LIN {X 0,Y 566.216,Z 387.456,A -85,B 0,C 180,E1 -2672.661,E2 -2672.661} C_VEL
LIN {X 0,Y 566.231,Z 387.453,A -85,B 0,C 180,E1 -2675.038,E2 -2675.038} C_VEL
LIN {X 0,Y 566.19,Z 387.454,A -85,B 0,C 180,E1 -2678.137,E2 -2678.137} C_VEL
LIN {X 0,Y 566.23,Z 387.456,A -85,B 0,C 180,E1 -2680.611,E2 -2680.611} C_VEL
LIN {X 0,Y 566.216,Z 387.449,A -85,B 0,C 180,E1 -2683.412,E2 -2683.412} C_VEL
LIN {X 0,Y 566.196,Z 387.457,A -85,B 0,C 180,E1 -2686.358,E2 -2686.358} C_VEL
LIN {X 0,Y 566.228,Z 387.456,A -85,B 0,C 180,E1 -2688.675,E2 -2688.675} C_VEL
LIN {X 0,Y 566.229,Z 387.447,A -85,B 0,C 180,E1 -2691.434,E2 -2691.434} C_VEL
LIN {X 0,Y 566.256,Z 387.451,A -85,B 0,C 180,E1 -2694.301,E2 -2694.301} C_VEL
LIN {X 0,Y 566.275,Z 387.444,A -85,B 0,C 180,E1 -2697.866,E2 -2697.866} C_VEL
LIN {X 0,Y 566.299,Z 387.443,A -85,B 0,C 180,E1 -2700.711,E2 -2700.711} C_VEL
LIN {X 0,Y 566.27,Z 387.445,A -85,B 0,C 180,E1 -2702.845,E2 -2702.845} C_VEL
LIN {X 0,Y 566.256,Z 387.446,A -85,B 0,C 180,E1 -2705.698,E2 -2705.698} C_VEL
LIN {X 0,Y 566.228,Z 387.452,A -85,B 0,C 180,E1 -2708.565,E2 -2708.565} C_VEL
LIN {X 0,Y 566.234,Z 387.447,A -85,B 0,C 180,E1 -2711.454,E2 -2711.454} C_VEL
LIN {X 0,Y 566.227,Z 387.452,A -85,B 0,C 180,E1 -2714.507,E2 -2714.507} C_VEL
LIN {X 0,Y 566.197,Z 387.452,A -85,B 0,C 180,E1 -2717.331,E2 -2717.331} C_VEL
LIN {X 0,Y 566.207,Z 387.456,A -85,B 0,C 180,E1 -2720.337,E2 -2720.337} C_VEL
LIN {X 0,Y 566.182,Z 387.455,A -85,B 0,C 180,E1 -2723.404,E2 -2723.404} C_VEL
LIN {X 0,Y 566.217,Z 387.455,A -85,B 0,C 180,E1 -2725.748,E2 -2725.748} C_VEL
LIN {X 0,Y 566.211,Z 387.451,A -85,B 0,C 180,E1 -2727.49,E2 -2727.49} C_VEL
LIN {X 0,Y 565.532,Z 387.542,A -85,B 0,C 180,E1 -2728.084,E2 -2728.084} C_VEL
LIN {X 0,Y 562.666,Z 387.896,A -85,B 0,C 180,E1 -2729.047,E2 -2729.047} C_VEL
LIN {X 0,Y 560.255,Z 388.2,A -85,B 0,C 180,E1 -2729.823,E2 -2729.823} C_VEL
LIN {X 0,Y 559.226,Z 388.322,A -85,B 0,C 180,E1 -2730.422,E2 -2730.422} C_VEL
LIN {X 0,Y 559.145,Z 388.331,A -85,B 0,C 180,E1 -2730.624,E2 -2730.624} C_VEL
LIN {X 0,Y 559.171,Z 388.332,A -85,B 0,C 180,E1 -2733.574,E2 -2733.574} C_VEL
LIN {X 0,Y 559.162,Z 388.329,A -85,B 0,C 180,E1 -2736.449,E2 -2736.449} C_VEL
LIN {X 0,Y 559.172,Z 388.327,A -85,B 0,C 180,E1 -2738.934,E2 -2738.934} C_VEL
LIN {X 0,Y 559.185,Z 388.335,A -85,B 0,C 180,E1 -2741.768,E2 -2741.768} C_VEL
LIN {X 0,Y 559.133,Z 388.331,A -85,B 0,C 180,E1 -2744.739,E2 -2744.739} C_VEL
LIN {X 0,Y 559.161,Z 388.331,A -85,B 0,C 180,E1 -2747.258,E2 -2747.258} C_VEL
LIN {X 0,Y 559.179,Z 388.328,A -85,B 0,C 180,E1 -2750.135,E2 -2750.135} C_VEL
LIN {X 0,Y 559.14,Z 388.331,A -85,B 0,C 180,E1 -2752.892,E2 -2752.892} C_VEL
LIN {X 0,Y 559.155,Z 388.338,A -85,B 0,C 180,E1 -2755.557,E2 -2755.557} C_VEL
LIN {X 0,Y 559.166,Z 388.328,A -85,B 0,C 180,E1 -2758.138,E2 -2758.138} C_VEL
LIN {X 0,Y 559.139,Z 388.331,A -85,B 0,C 180,E1 -2760.647,E2 -2760.647} C_VEL
LIN {X 0,Y 559.177,Z 388.332,A -85,B 0,C 180,E1 -2763.17,E2 -2763.17} C_VEL
LIN {X 0,Y 559.153,Z 388.337,A -85,B 0,C 180,E1 -2765.495,E2 -2765.495} C_VEL
LIN {X 0,Y 559.167,Z 388.328,A -85,B 0,C 180,E1 -2768.624,E2 -2768.624} C_VEL
LIN {X 0,Y 559.165,Z 388.331,A -85,B 0,C 180,E1 -2770.927,E2 -2770.927} C_VEL
LIN {X 0,Y 559.163,Z 388.33,A -85,B 0,C 180,E1 -2773.948,E2 -2773.948} C_VEL
LIN {X 0,Y 559.169,Z 388.328,A -85,B 0,C 180,E1 -2776.184,E2 -2776.184} C_VEL
LIN {X 0,Y 559.193,Z 388.334,A -85,B 0,C 180,E1 -2779.134,E2 -2779.134} C_VEL
LIN {X 0,Y 559.203,Z 388.324,A -85,B 0,C 180,E1 -2782.054,E2 -2782.054} C_VEL
LIN {X 0,Y 559.253,Z 388.325,A -85,B 0,C 180,E1 -2784.954,E2 -2784.954} C_VEL
LIN {X 0,Y 559.254,Z 388.318,A -85,B 0,C 180,E1 -2787.84,E2 -2787.84} C_VEL
LIN {X 0,Y 559.27,Z 388.321,A -85,B 0,C 180,E1 -2790.72,E2 -2790.72} C_VEL
LIN {X 0,Y 559.236,Z 388.328,A -85,B 0,C 180,E1 -2792.882,E2 -2792.882} C_VEL
LIN {X 0,Y 559.236,Z 388.32,A -85,B 0,C 180,E1 -2795.77,E2 -2795.77} C_VEL
LIN {X 0,Y 559.189,Z 388.332,A -85,B 0,C 180,E1 -2798.674,E2 -2798.674} C_VEL
LIN {X 0,Y 559.202,Z 388.324,A -85,B 0,C 180,E1 -2801.6,E2 -2801.6} C_VEL
LIN {X 0,Y 559.197,Z 388.331,A -85,B 0,C 180,E1 -2804.596,E2 -2804.596} C_VEL
LIN {X 0,Y 559.156,Z 388.33,A -85,B 0,C 180,E1 -2807.557,E2 -2807.557} C_VEL
LIN {X 0,Y 559.169,Z 388.327,A -85,B 0,C 180,E1 -2809.837,E2 -2809.837} C_VEL
LIN {X 0,Y 559.139,Z 388.333,A -85,B 0,C 180,E1 -2812.153,E2 -2812.153} C_VEL
LIN {X 0,Y 559.176,Z 388.328,A -85,B 0,C 180,E1 -2815.187,E2 -2815.187} C_VEL
LIN {X 0,Y 559.191,Z 388.324,A -85,B 0,C 180,E1 -2817.711,E2 -2817.711} C_VEL
LIN {X 0,Y 559.159,Z 388.331,A -85,B 0,C 180,E1 -2821.019,E2 -2821.019} C_VEL
LIN {X 0,Y 559.163,Z 388.33,A -85,B 0,C 180,E1 -2823.949,E2 -2823.949} C_VEL
LIN {X 0,Y 559.185,Z 388.335,A -85,B 0,C 180,E1 -2826.451,E2 -2826.451} C_VEL
LIN {X 0,Y 559.173,Z 388.328,A -85,B 0,C 180,E1 -2828.934,E2 -2828.934} C_VEL
LIN {X 0,Y 559.188,Z 388.326,A -85,B 0,C 180,E1 -2831.767,E2 -2831.767} C_VEL
LIN {X 0,Y 559.135,Z 388.334,A -85,B 0,C 180,E1 -2834.739,E2 -2834.739} C_VEL
LIN {X 0,Y 559.156,Z 388.328,A -85,B 0,C 180,E1 -2837.257,E2 -2837.257} C_VEL
LIN {X 0,Y 559.181,Z 388.334,A -85,B 0,C 180,E1 -2840.135,E2 -2840.135} C_VEL
LIN {X 0,Y 559.142,Z 388.331,A -85,B 0,C 180,E1 -2842.892,E2 -2842.892} C_VEL
LIN {X 0,Y 559.152,Z 388.331,A -85,B 0,C 180,E1 -2845.556,E2 -2845.556} C_VEL
LIN {X 0,Y 559.165,Z 388.337,A -85,B 0,C 180,E1 -2848.138,E2 -2848.138} C_VEL
LIN {X 0,Y 559.152,Z 388.331,A -85,B 0,C 180,E1 -2850.647,E2 -2850.647} C_VEL
LIN {X 0,Y 559.167,Z 388.327,A -85,B 0,C 180,E1 -2853.172,E2 -2853.172} C_VEL
LIN {X 0,Y 559.152,Z 388.332,A -85,B 0,C 180,E1 -2855.495,E2 -2855.495} C_VEL
LIN {X 0,Y 559.166,Z 388.328,A -85,B 0,C 180,E1 -2858.624,E2 -2858.624} C_VEL
LIN {X 0,Y 559.166,Z 388.327,A -85,B 0,C 180,E1 -2860.927,E2 -2860.927} C_VEL
LIN {X 0,Y 559.167,Z 388.336,A -85,B 0,C 180,E1 -2863.948,E2 -2863.948} C_VEL
LIN {X 0,Y 559.17,Z 388.331,A -85,B 0,C 180,E1 -2866.184,E2 -2866.184} C_VEL
LIN {X 0,Y 559.19,Z 388.325,A -85,B 0,C 180,E1 -2869.134,E2 -2869.134} C_VEL
LIN {X 0,Y 559.203,Z 388.327,A -85,B 0,C 180,E1 -2872.054,E2 -2872.054} C_VEL
LIN {X 0,Y 559.252,Z 388.317,A -85,B 0,C 180,E1 -2874.954,E2 -2874.954} C_VEL
LIN {X 0,Y 559.248,Z 388.324,A -85,B 0,C 180,E1 -2877.84,E2 -2877.84} C_VEL
LIN {X 0,Y 559.27,Z 388.314,A -85,B 0,C 180,E1 -2880.72,E2 -2880.72} C_VEL
LIN {X 0,Y 559.238,Z 388.319,A -85,B 0,C 180,E1 -2882.882,E2 -2882.882} C_VEL
LIN {X 0,Y 559.227,Z 388.325,A -85,B 0,C 180,E1 -2885.771,E2 -2885.771} C_VEL
LIN {X 0,Y 559.189,Z 388.325,A -85,B 0,C 180,E1 -2888.675,E2 -2888.675} C_VEL
LIN {X 0,Y 559.202,Z 388.33,A -85,B 0,C 180,E1 -2891.601,E2 -2891.601} C_VEL
LIN {X 0,Y 559.196,Z 388.324,A -85,B 0,C 180,E1 -2894.596,E2 -2894.596} C_VEL
LIN {X 0,Y 559.16,Z 388.334,A -85,B 0,C 180,E1 -2897.557,E2 -2897.557} C_VEL
LIN {X 0,Y 559.17,Z 388.329,A -85,B 0,C 180,E1 -2899.838,E2 -2899.838} C_VEL
LIN {X 0,Y 559.139,Z 388.331,A -85,B 0,C 180,E1 -2902.153,E2 -2902.153} C_VEL
LIN {X 0,Y 559.177,Z 388.335,A -85,B 0,C 180,E1 -2905.188,E2 -2905.188} C_VEL
LIN {X 0,Y 559.187,Z 388.327,A -85,B 0,C 180,E1 -2907.712,E2 -2907.712} C_VEL
LIN {X 0,Y 559.155,Z 388.329,A -85,B 0,C 180,E1 -2910.183,E2 -2910.183} C_VEL
LIN {X 0,Y 559.174,Z 388.33,A -85,B 0,C 180,E1 -2912.714,E2 -2912.714} C_VEL
LIN {X 0,Y 559.157,Z 388.335,A -85,B 0,C 180,E1 -2915.322,E2 -2915.322} C_VEL
LIN {X 0,Y 559.135,Z 388.333,A -85,B 0,C 180,E1 -2918.018,E2 -2918.018} C_VEL
LIN {X 0,Y 559.176,Z 388.335,A -85,B 0,C 180,E1 -2920.811,E2 -2920.811} C_VEL
LIN {X 0,Y 559.141,Z 388.335,A -85,B 0,C 180,E1 -2923.734,E2 -2923.734} C_VEL
LIN {X 0,Y 559.154,Z 388.337,A -85,B 0,C 180,E1 -2926.268,E2 -2926.268} C_VEL
LIN {X 0,Y 559.57,Z 391.187,A -85,B 0,C 180,E1 -2928.267,E2 -2928.267} C_VEL
LIN {X 0,Y 559.531,Z 394.347,A -85,B 0,C 180,E1 -2930.165,E2 -2930.165} C_VEL
LIN {X 0,Y 559.375,Z 399.291,A -85,B 0,C 180,E1 -2932.91,E2 -2932.91} C_VEL
LIN {X 0,Y 559.267,Z 404.344,A -85,B 0,C 180,E1 -2935.564,E2 -2935.564} C_VEL
LIN {X 0,Y 559.208,Z 409.734,A -85,B 0,C 180,E1 -2938.14,E2 -2938.14} C_VEL
LIN {X 0,Y 559.125,Z 415.123,A -85,B 0,C 180,E1 -2940.646,E2 -2940.646} C_VEL
LIN {X 0,Y 559.091,Z 420.725,A -85,B 0,C 180,E1 -2943.189,E2 -2943.189} C_VEL
LIN {X 0,Y 559.022,Z 425.902,A -85,B 0,C 180,E1 -2945.489,E2 -2945.489} C_VEL
LIN {X 0,Y 559.006,Z 432.793,A -85,B 0,C 180,E1 -2948.49,E2 -2948.49} C_VEL
LIN {X 0,Y 558.952,Z 438.478,A -85,B 0,C 180,E1 -2950.919,E2 -2950.919} C_VEL
LIN {X 0,Y 558.889,Z 443.867,A -85,B 0,C 180,E1 -2953.189,E2 -2953.189} C_VEL
LIN {X 0,Y 558.852,Z 451.053,A -85,B 0,C 180,E1 -2956.176,E2 -2956.176} C_VEL
LIN {X 0,Y 558.849,Z 453.523,A -85,B 0,C 180,E1 -2957.194,E2 -2957.194} C_VEL
LIN {X 0,Y 559.976,Z 461.405,A -85,B 0,C 180,E1 -2957.382,E2 -2957.382} C_VEL
LIN {X 0,Y 559.871,Z 473.243,A -85,B 0,C 180,E1 -2957.729,E2 -2957.729} C_VEL
LIN {X 0,Y 559.731,Z 484.244,A -85,B 0,C 180,E1 -2958.171,E2 -2958.171} C_VEL
LIN {X 0,Y 559.607,Z 495.133,A -85,B 0,C 180,E1 -2958.738,E2 -2958.738} C_VEL
LIN {X 0,Y 559.427,Z 506.748,A -85,B 0,C 180,E1 -2959.504,E2 -2959.504} C_VEL
LIN {X 0,Y 559.297,Z 515.638,A -85,B 0,C 180,E1 -2960.233,E2 -2960.233} C_VEL
LIN {X 0,Y 559.141,Z 524.76,A -85,B 0,C 180,E1 -2961.143,E2 -2961.143} C_VEL
LIN {X 0,Y 559.053,Z 532.307,A -85,B 0,C 180,E1 -2962.051,E2 -2962.051} C_VEL
LIN {X 0,Y 558.923,Z 539.955,A -85,B 0,C 180,E1 -2963.176,E2 -2963.176} C_VEL
LIN {X 0,Y 558.929,Z 545.682,A -85,B 0,C 180,E1 -2964.227,E2 -2964.227} C_VEL
LIN {X 0,Y 558.826,Z 550.378,A -85,B 0,C 180,E1 -2965.311,E2 -2965.311} C_VEL
LIN {X 0,Y 558.836,Z 553.965,A -85,B 0,C 180,E1 -2966.395,E2 -2966.395} C_VEL
LIN {X 0,Y 558.799,Z 555.792,A -85,B 0,C 180,E1 -2967.116,E2 -2967.116} C_VEL
LIN {X 0,Y 558.746,Z 558.189,A -85,B 0,C 180,E1 -2968.558,E2 -2968.558} C_VEL
LIN {X 0,Y 558.741,Z 558.782,A -85,B 0,C 180,E1 -2969.279,E2 -2969.279} C_VEL
LIN {X 0,Y 558.741,Z 558.782,A -85,B 0,C 180,E1 -2970.721,E2 -2970.721} C_VEL
LIN {X 0,Y 558.746,Z 558.19,A -85,B 0,C 180,E1 -2971.441,E2 -2971.441} C_VEL
LIN {X 0,Y 558.799,Z 555.793,A -85,B 0,C 180,E1 -2972.883,E2 -2972.883} C_VEL
LIN {X 0,Y 558.844,Z 552.88,A -85,B 0,C 180,E1 -2973.966,E2 -2973.966} C_VEL
LIN {X 0,Y 558.798,Z 548.931,A -85,B 0,C 180,E1 -2975.051,E2 -2975.051} C_VEL
LIN {X 0,Y 558.909,Z 543.836,A -85,B 0,C 180,E1 -2976.135,E2 -2976.135} C_VEL
LIN {X 0,Y 558.974,Z 537.453,A -85,B 0,C 180,E1 -2977.223,E2 -2977.223} C_VEL
LIN {X 0,Y 559.099,Z 529.492,A -85,B 0,C 180,E1 -2978.311,E2 -2978.311} C_VEL
LIN {X 0,Y 559.207,Z 521.351,A -85,B 0,C 180,E1 -2979.22,E2 -2979.22} C_VEL
LIN {X 0,Y 559.359,Z 511.359,A -85,B 0,C 180,E1 -2980.131,E2 -2980.131} C_VEL
LIN {X 0,Y 559.531,Z 501.541,A -85,B 0,C 180,E1 -2980.86,E2 -2980.86} C_VEL
LIN {X 0,Y 559.63,Z 490.288,A -85,B 0,C 180,E1 -2981.534,E2 -2981.534} C_VEL
LIN {X 0,Y 559.828,Z 476.988,A -85,B 0,C 180,E1 -2982.138,E2 -2982.138} C_VEL
LIN {X 0,Y 559.963,Z 464.987,A -85,B 0,C 180,E1 -2982.526,E2 -2982.526} C_VEL
LIN {X 0,Y 559.737,Z 458.848,A -85,B 0,C 180,E1 -2982.684,E2 -2982.684} C_VEL
LIN {X 0,Y 558.849,Z 453.524,A -85,B 0,C 180,E1 -2982.806,E2 -2982.806} C_VEL
LIN {X 0,Y 558.869,Z 447.461,A -85,B 0,C 180,E1 -2985.312,E2 -2985.312} C_VEL
LIN {X 0,Y 558.922,Z 440.275,A -85,B 0,C 180,E1 -2988.321,E2 -2988.321} C_VEL
LIN {X 0,Y 558.947,Z 434.885,A -85,B 0,C 180,E1 -2990.613,E2 -2990.613} C_VEL
LIN {X 0,Y 559.028,Z 428.432,A -85,B 0,C 180,E1 -2993.401,E2 -2993.401} C_VEL
LIN {X 0,Y 559.069,Z 422.31,A -85,B 0,C 180,E1 -2996.102,E2 -2996.102} C_VEL
LIN {X 0,Y 559.113,Z 416.92,A -85,B 0,C 180,E1 -2998.532,E2 -2998.532} C_VEL
LIN {X 0,Y 559.184,Z 410.971,A -85,B 0,C 180,E1 -3001.279,E2 -3001.279} C_VEL
LIN {X 0,Y 559.269,Z 405.317,A -85,B 0,C 180,E1 -3003.964,E2 -3003.964} C_VEL
LIN {X 0,Y 559.361,Z 400.43,A -85,B 0,C 180,E1 -3006.474,E2 -3006.474} C_VEL
LIN {X 0,Y 559.509,Z 395.979,A -85,B 0,C 180,E1 -3008.906,E2 -3008.906} C_VEL
LIN {X 0,Y 559.606,Z 392.177,A -85,B 0,C 180,E1 -3011.102,E2 -3011.102} C_VEL
LIN {X 0,Y 559.227,Z 388.907,A -85,B 0,C 180,E1 -3013.205,E2 -3013.205} C_VEL
LIN {X 0,Y 559.152,Z 388.336,A -85,B 0,C 180,E1 -3013.732,E2 -3013.732} C_VEL
LIN {X 0,Y 559.144,Z 388.338,A -85,B 0,C 180,E1 -3016.803,E2 -3016.803} C_VEL
LIN {X 0,Y 559.174,Z 388.335,A -85,B 0,C 180,E1 -3019.189,E2 -3019.189} C_VEL
LIN {X 0,Y 559.133,Z 388.333,A -85,B 0,C 180,E1 -3021.982,E2 -3021.982} C_VEL
LIN {X 0,Y 559.157,Z 388.337,A -85,B 0,C 180,E1 -3024.782,E2 -3024.782} C_VEL
LIN {X 0,Y 559.17,Z 388.33,A -85,B 0,C 180,E1 -3027.361,E2 -3027.361} C_VEL
LIN {X 0,Y 559.185,Z 388.326,A -85,B 0,C 180,E1 -3030.134,E2 -3030.134} C_VEL
LIN {X 0,Y 559.168,Z 388.331,A -85,B 0,C 180,E1 -3033.171,E2 -3033.171} C_VEL
LIN {X 0,Y 559.152,Z 388.33,A -85,B 0,C 180,E1 -3035.494,E2 -3035.494} C_VEL
LIN {X 0,Y 559.166,Z 388.336,A -85,B 0,C 180,E1 -3038.623,E2 -3038.623} C_VEL
LIN {X 0,Y 559.166,Z 388.333,A -85,B 0,C 180,E1 -3040.926,E2 -3040.926} C_VEL
LIN {X 0,Y 559.166,Z 388.328,A -85,B 0,C 180,E1 -3043.948,E2 -3043.948} C_VEL
LIN {X 0,Y 559.17,Z 388.33,A -85,B 0,C 180,E1 -3046.184,E2 -3046.184} C_VEL
LIN {X 0,Y 559.189,Z 388.326,A -85,B 0,C 180,E1 -3049.133,E2 -3049.133} C_VEL
LIN {X 0,Y 559.201,Z 388.326,A -85,B 0,C 180,E1 -3052.053,E2 -3052.053} C_VEL
LIN {X 0,Y 559.251,Z 388.319,A -85,B 0,C 180,E1 -3054.953,E2 -3054.953} C_VEL
LIN {X 0,Y 559.247,Z 388.319,A -85,B 0,C 180,E1 -3057.839,E2 -3057.839} C_VEL
LIN {X 0,Y 559.269,Z 388.319,A -85,B 0,C 180,E1 -3060.72,E2 -3060.72} C_VEL
LIN {X 0,Y 559.236,Z 388.321,A -85,B 0,C 180,E1 -3062.881,E2 -3062.881} C_VEL
LIN {X 0,Y 559.225,Z 388.322,A -85,B 0,C 180,E1 -3065.77,E2 -3065.77} C_VEL
LIN {X 0,Y 559.187,Z 388.328,A -85,B 0,C 180,E1 -3068.674,E2 -3068.674} C_VEL
LIN {X 0,Y 559.198,Z 388.325,A -85,B 0,C 180,E1 -3071.6,E2 -3071.6} C_VEL
LIN {X 0,Y 559.191,Z 388.327,A -85,B 0,C 180,E1 -3074.595,E2 -3074.595} C_VEL
LIN {X 0,Y 559.157,Z 388.33,A -85,B 0,C 180,E1 -3077.557,E2 -3077.557} C_VEL
LIN {X 0,Y 559.165,Z 388.333,A -85,B 0,C 180,E1 -3079.837,E2 -3079.837} C_VEL
LIN {X 0,Y 559.134,Z 388.339,A -85,B 0,C 180,E1 -3082.153,E2 -3082.153} C_VEL
LIN {X 0,Y 559.172,Z 388.327,A -85,B 0,C 180,E1 -3085.187,E2 -3085.187} C_VEL
LIN {X 0,Y 559.188,Z 388.33,A -85,B 0,C 180,E1 -3087.711,E2 -3087.711} C_VEL
LIN {X 0,Y 559.145,Z 388.331,A -85,B 0,C 180,E1 -3090.624,E2 -3090.624} C_VEL
LIN {X 0,Y 558.482,Z 388.414,A -85,B 0,C 180,E1 -3091.226,E2 -3091.226} C_VEL
LIN {X 0,Y 555.619,Z 388.774,A -85,B 0,C 180,E1 -3092.202,E2 -3092.202} C_VEL
LIN {X 0,Y 553.208,Z 389.071,A -85,B 0,C 180,E1 -3092.988,E2 -3092.988} C_VEL
LIN {X 0,Y 552.19,Z 389.202,A -85,B 0,C 180,E1 -3093.594,E2 -3093.594} C_VEL
LIN {X 0,Y 552.116,Z 389.209,A -85,B 0,C 180,E1 -3093.8,E2 -3093.8} C_VEL
LIN {X 0,Y 552.105,Z 389.207,A -85,B 0,C 180,E1 -3096.747,E2 -3096.747} C_VEL
LIN {X 0,Y 552.128,Z 389.21,A -85,B 0,C 180,E1 -3099.527,E2 -3099.527} C_VEL
LIN {X 0,Y 552.123,Z 389.205,A -85,B 0,C 180,E1 -3102.425,E2 -3102.425} C_VEL
LIN {X 0,Y 552.093,Z 389.216,A -85,B 0,C 180,E1 -3105.563,E2 -3105.563} C_VEL
LIN {X 0,Y 552.134,Z 389.203,A -85,B 0,C 180,E1 -3108.676,E2 -3108.676} C_VEL
LIN {X 0,Y 552.114,Z 389.212,A -85,B 0,C 180,E1 -3111.412,E2 -3111.412} C_VEL
LIN {X 0,Y 552.107,Z 389.208,A -85,B 0,C 180,E1 -3114.159,E2 -3114.159} C_VEL
LIN {X 0,Y 552.124,Z 389.205,A -85,B 0,C 180,E1 -3116.815,E2 -3116.815} C_VEL
LIN {X 0,Y 552.102,Z 389.216,A -85,B 0,C 180,E1 -3119.391,E2 -3119.391} C_VEL
LIN {X 0,Y 552.122,Z 389.208,A -85,B 0,C 180,E1 -3121.903,E2 -3121.903} C_VEL
LIN {X 0,Y 552.152,Z 389.202,A -85,B 0,C 180,E1 -3124.649,E2 -3124.649} C_VEL
LIN {X 0,Y 552.092,Z 389.215,A -85,B 0,C 180,E1 -3127.55,E2 -3127.55} C_VEL
LIN {X 0,Y 552.144,Z 389.202,A -85,B 0,C 180,E1 -3130.374,E2 -3130.374} C_VEL
LIN {X 0,Y 552.151,Z 389.207,A -85,B 0,C 180,E1 -3132.978,E2 -3132.978} C_VEL
LIN {X 0,Y 552.132,Z 389.205,A -85,B 0,C 180,E1 -3136.005,E2 -3136.005} C_VEL
LIN {X 0,Y 552.16,Z 389.208,A -85,B 0,C 180,E1 -3138.994,E2 -3138.994} C_VEL
LIN {X 0,Y 552.157,Z 389.202,A -85,B 0,C 180,E1 -3141.952,E2 -3141.952} C_VEL
LIN {X 0,Y 552.228,Z 389.199,A -85,B 0,C 180,E1 -3144.889,E2 -3144.889} C_VEL
LIN {X 0,Y 552.225,Z 389.194,A -85,B 0,C 180,E1 -3147.812,E2 -3147.812} C_VEL
LIN {X 0,Y 552.24,Z 389.197,A -85,B 0,C 180,E1 -3150.729,E2 -3150.729} C_VEL
LIN {X 0,Y 552.202,Z 389.204,A -85,B 0,C 180,E1 -3152.918,E2 -3152.918} C_VEL
LIN {X 0,Y 552.207,Z 389.196,A -85,B 0,C 180,E1 -3155.844,E2 -3155.844} C_VEL
LIN {X 0,Y 552.16,Z 389.209,A -85,B 0,C 180,E1 -3158.786,E2 -3158.786} C_VEL
LIN {X 0,Y 552.16,Z 389.201,A -85,B 0,C 180,E1 -3161.751,E2 -3161.751} C_VEL
LIN {X 0,Y 552.134,Z 389.213,A -85,B 0,C 180,E1 -3164.748,E2 -3164.748} C_VEL
LIN {X 0,Y 552.108,Z 389.208,A -85,B 0,C 180,E1 -3167.788,E2 -3167.788} C_VEL
LIN {X 0,Y 552.128,Z 389.206,A -85,B 0,C 180,E1 -3170.101,E2 -3170.101} C_VEL
LIN {X 0,Y 552.093,Z 389.215,A -85,B 0,C 180,E1 -3172.451,E2 -3172.451} C_VEL
LIN {X 0,Y 552.154,Z 389.201,A -85,B 0,C 180,E1 -3175.351,E2 -3175.351} C_VEL
LIN {X 0,Y 552.123,Z 389.207,A -85,B 0,C 180,E1 -3178.097,E2 -3178.097} C_VEL
LIN {X 0,Y 552.103,Z 389.216,A -85,B 0,C 180,E1 -3180.609,E2 -3180.609} C_VEL
LIN {X 0,Y 552.119,Z 389.206,A -85,B 0,C 180,E1 -3183.185,E2 -3183.185} C_VEL
LIN {X 0,Y 552.109,Z 389.208,A -85,B 0,C 180,E1 -3185.842,E2 -3185.842} C_VEL
LIN {X 0,Y 552.121,Z 389.206,A -85,B 0,C 180,E1 -3189.062,E2 -3189.062} C_VEL
LIN {X 0,Y 552.136,Z 389.203,A -85,B 0,C 180,E1 -3191.444,E2 -3191.444} C_VEL
LIN {X 0,Y 552.092,Z 389.215,A -85,B 0,C 180,E1 -3194.532,E2 -3194.532} C_VEL
LIN {X 0,Y 552.126,Z 389.205,A -85,B 0,C 180,E1 -3197.585,E2 -3197.585} C_VEL
LIN {X 0,Y 552.13,Z 389.209,A -85,B 0,C 180,E1 -3200.473,E2 -3200.473} C_VEL
LIN {X 0,Y 552.11,Z 389.206,A -85,B 0,C 180,E1 -3203.316,E2 -3203.316} C_VEL
LIN {X 0,Y 552.126,Z 389.211,A -85,B 0,C 180,E1 -3205.94,E2 -3205.94} C_VEL
LIN {X 0,Y 552.113,Z 389.209,A -85,B 0,C 180,E1 -3208.541,E2 -3208.541} C_VEL
LIN {X 0,Y 552.121,Z 389.206,A -85,B 0,C 180,E1 -3211.438,E2 -3211.438} C_VEL
LIN {X 0,Y 552.125,Z 389.209,A -85,B 0,C 180,E1 -3214.356,E2 -3214.356} C_VEL
LIN {X 0,Y 552.105,Z 389.207,A -85,B 0,C 180,E1 -3216.759,E2 -3216.759} C_VEL
LIN {X 0,Y 552.115,Z 389.206,A -85,B 0,C 180,E1 -3219.12,E2 -3219.12} C_VEL
LIN {X 0,Y 552.126,Z 389.207,A -85,B 0,C 180,E1 -3221.445,E2 -3221.445} C_VEL
LIN {X 0,Y 552.117,Z 389.213,A -85,B 0,C 180,E1 -3223.738,E2 -3223.738} C_VEL
LIN {X 0,Y 552.133,Z 389.21,A -85,B 0,C 180,E1 -3226.005,E2 -3226.005} C_VEL
LIN {X 0,Y 552.158,Z 389.201,A -85,B 0,C 180,E1 -3228.994,E2 -3228.994} C_VEL
LIN {X 0,Y 552.156,Z 389.207,A -85,B 0,C 180,E1 -3231.952,E2 -3231.952} C_VEL
LIN {X 0,Y 552.226,Z 389.192,A -85,B 0,C 180,E1 -3234.889,E2 -3234.889} C_VEL
LIN {X 0,Y 552.219,Z 389.2,A -85,B 0,C 180,E1 -3237.812,E2 -3237.812} C_VEL
LIN {X 0,Y 552.24,Z 389.19,A -85,B 0,C 180,E1 -3240.73,E2 -3240.73} C_VEL
LIN {X 0,Y 552.204,Z 389.196,A -85,B 0,C 180,E1 -3242.919,E2 -3242.919} C_VEL
LIN {X 0,Y 552.197,Z 389.2,A -85,B 0,C 180,E1 -3245.844,E2 -3245.844} C_VEL
LIN {X 0,Y 552.16,Z 389.201,A -85,B 0,C 180,E1 -3248.786,E2 -3248.786} C_VEL
LIN {X 0,Y 552.159,Z 389.205,A -85,B 0,C 180,E1 -3251.751,E2 -3251.751} C_VEL
LIN {X 0,Y 552.133,Z 389.205,A -85,B 0,C 180,E1 -3254.749,E2 -3254.749} C_VEL
LIN {X 0,Y 552.112,Z 389.209,A -85,B 0,C 180,E1 -3257.789,E2 -3257.789} C_VEL
LIN {X 0,Y 552.128,Z 389.204,A -85,B 0,C 180,E1 -3260.102,E2 -3260.102} C_VEL
LIN {X 0,Y 552.094,Z 389.209,A -85,B 0,C 180,E1 -3262.451,E2 -3262.451} C_VEL
LIN {X 0,Y 552.153,Z 389.208,A -85,B 0,C 180,E1 -3265.351,E2 -3265.351} C_VEL
LIN {X 0,Y 552.121,Z 389.205,A -85,B 0,C 180,E1 -3268.098,E2 -3268.098} C_VEL
LIN {X 0,Y 552.106,Z 389.209,A -85,B 0,C 180,E1 -3270.609,E2 -3270.609} C_VEL
LIN {X 0,Y 552.122,Z 389.214,A -85,B 0,C 180,E1 -3273.186,E2 -3273.186} C_VEL
LIN {X 0,Y 552.113,Z 389.207,A -85,B 0,C 180,E1 -3275.842,E2 -3275.842} C_VEL
LIN {X 0,Y 552.126,Z 389.214,A -85,B 0,C 180,E1 -3279.063,E2 -3279.063} C_VEL
LIN {X 0,Y 552.14,Z 389.208,A -85,B 0,C 180,E1 -3281.445,E2 -3281.445} C_VEL
LIN {X 0,Y 552.095,Z 389.216,A -85,B 0,C 180,E1 -3284.532,E2 -3284.532} C_VEL
LIN {X 0,Y 552.1,Z 389.215,A -85,B 0,C 180,E1 -3285.563,E2 -3285.563} C_VEL
LIN {X 0,Y 552.2,Z 389.903,A -85,B 0,C 180,E1 -3286.586,E2 -3286.586} C_VEL
LIN {X 0,Y 552.631,Z 393.024,A -85,B 0,C 180,E1 -3288.619,E2 -3288.619} C_VEL
LIN {X 0,Y 552.483,Z 397.791,A -85,B 0,C 180,E1 -3291.442,E2 -3291.442} C_VEL
LIN {X 0,Y 552.298,Z 403.428,A -85,B 0,C 180,E1 -3294.529,E2 -3294.529} C_VEL
LIN {X 0,Y 552.214,Z 408.592,A -85,B 0,C 180,E1 -3297.138,E2 -3297.138} C_VEL
LIN {X 0,Y 552.124,Z 415.123,A -85,B 0,C 180,E1 -3300.236,E2 -3300.236} C_VEL
LIN {X 0,Y 552.045,Z 421.165,A -85,B 0,C 180,E1 -3303.02,E2 -3303.02} C_VEL
LIN {X 0,Y 551.978,Z 425.902,A -85,B 0,C 180,E1 -3305.155,E2 -3305.155} C_VEL
LIN {X 0,Y 551.92,Z 431.292,A -85,B 0,C 180,E1 -3307.542,E2 -3307.542} C_VEL
LIN {X 0,Y 551.886,Z 438.478,A -85,B 0,C 180,E1 -3310.665,E2 -3310.665} C_VEL
LIN {X 0,Y 551.784,Z 445.664,A -85,B 0,C 180,E1 -3313.727,E2 -3313.727} C_VEL
LIN {X 0,Y 551.764,Z 451.053,A -85,B 0,C 180,E1 -3315.995,E2 -3315.995} C_VEL
LIN {X 0,Y 551.746,Z 453.523,A -85,B 0,C 180,E1 -3317.026,E2 -3317.026} C_VEL
LIN {X 0,Y 553.041,Z 462.315,A -85,B 0,C 180,E1 -3317.244,E2 -3317.244} C_VEL
LIN {X 0,Y 552.933,Z 474.394,A -85,B 0,C 180,E1 -3317.615,E2 -3317.615} C_VEL
LIN {X 0,Y 552.772,Z 485.445,A -85,B 0,C 180,E1 -3318.077,E2 -3318.077} C_VEL
LIN {X 0,Y 552.604,Z 496.95,A -85,B 0,C 180,E1 -3318.701,E2 -3318.701} C_VEL
LIN {X 0,Y 552.405,Z 507.918,A -85,B 0,C 180,E1 -3319.462,E2 -3319.462} C_VEL
LIN {X 0,Y 552.233,Z 517.576,A -85,B 0,C 180,E1 -3320.292,E2 -3320.292} C_VEL
LIN {X 0,Y 552.083,Z 526.379,A -85,B 0,C 180,E1 -3321.213,E2 -3321.213} C_VEL
LIN {X 0,Y 551.95,Z 535.007,A -85,B 0,C 180,E1 -3322.317,E2 -3322.317} C_VEL
LIN {X 0,Y 551.823,Z 541.872,A -85,B 0,C 180,E1 -3323.418,E2 -3323.418} C_VEL
LIN {X 0,Y 551.802,Z 547.363,A -85,B 0,C 180,E1 -3324.518,E2 -3324.518} C_VEL
LIN {X 0,Y 551.764,Z 551.662,A -85,B 0,C 180,E1 -3325.617,E2 -3325.617} C_VEL
LIN {X 0,Y 551.75,Z 553.967,A -85,B 0,C 180,E1 -3326.348,E2 -3326.348} C_VEL
LIN {X 0,Y 551.724,Z 555.789,A -85,B 0,C 180,E1 -3327.079,E2 -3327.079} C_VEL
LIN {X 0,Y 551.645,Z 558.19,A -85,B 0,C 180,E1 -3328.54,E2 -3328.54} C_VEL
LIN {X 0,Y 551.641,Z 558.781,A -85,B 0,C 180,E1 -3329.27,E2 -3329.27} C_VEL
LIN {X 0,Y 551.641,Z 558.782,A -85,B 0,C 180,E1 -3330.73,E2 -3330.73} C_VEL
LIN {X 0,Y 551.645,Z 558.191,A -85,B 0,C 180,E1 -3331.46,E2 -3331.46} C_VEL
LIN {X 0,Y 551.724,Z 555.79,A -85,B 0,C 180,E1 -3332.92,E2 -3332.92} C_VEL
LIN {X 0,Y 551.763,Z 552.876,A -85,B 0,C 180,E1 -3334.017,E2 -3334.017} C_VEL
LIN {X 0,Y 551.723,Z 548.926,A -85,B 0,C 180,E1 -3335.116,E2 -3335.116} C_VEL
LIN {X 0,Y 551.836,Z 544.436,A -85,B 0,C 180,E1 -3336.098,E2 -3336.098} C_VEL
LIN {X 0,Y 551.886,Z 538.598,A -85,B 0,C 180,E1 -3337.132,E2 -3337.132} C_VEL
LIN {X 0,Y 552.013,Z 530.936,A -85,B 0,C 180,E1 -3338.235,E2 -3338.235} C_VEL
LIN {X 0,Y 552.165,Z 521.353,A -85,B 0,C 180,E1 -3339.339,E2 -3339.339} C_VEL
LIN {X 0,Y 552.368,Z 511.353,A -85,B 0,C 180,E1 -3340.26,E2 -3340.26} C_VEL
LIN {X 0,Y 552.531,Z 501.533,A -85,B 0,C 180,E1 -3340.999,E2 -3340.999} C_VEL
LIN {X 0,Y 552.668,Z 491.034,A -85,B 0,C 180,E1 -3341.641,E2 -3341.641} C_VEL
LIN {X 0,Y 552.849,Z 478.154,A -85,B 0,C 180,E1 -3342.247,E2 -3342.247} C_VEL
LIN {X 0,Y 553.043,Z 465.844,A -85,B 0,C 180,E1 -3342.662,E2 -3342.662} C_VEL
LIN {X 0,Y 552.83,Z 459.981,A -85,B 0,C 180,E1 -3342.82,E2 -3342.82} C_VEL
LIN {X 0,Y 551.747,Z 453.524,A -85,B 0,C 180,E1 -3342.973,E2 -3342.973} C_VEL
LIN {X 0,Y 551.783,Z 447.461,A -85,B 0,C 180,E1 -3345.514,E2 -3345.514} C_VEL
LIN {X 0,Y 551.836,Z 442.071,A -85,B 0,C 180,E1 -3347.797,E2 -3347.797} C_VEL
LIN {X 0,Y 551.896,Z 436.682,A -85,B 0,C 180,E1 -3350.11,E2 -3350.11} C_VEL
LIN {X 0,Y 551.919,Z 431.292,A -85,B 0,C 180,E1 -3352.458,E2 -3352.458} C_VEL
LIN {X 0,Y 552.015,Z 424.841,A -85,B 0,C 180,E1 -3355.319,E2 -3355.319} C_VEL
LIN {X 0,Y 552.044,Z 418.717,A -85,B 0,C 180,E1 -3358.101,E2 -3358.101} C_VEL
LIN {X 0,Y 552.116,Z 413.327,A -85,B 0,C 180,E1 -3360.608,E2 -3360.608} C_VEL
LIN {X 0,Y 552.216,Z 407.938,A -85,B 0,C 180,E1 -3363.178,E2 -3363.178} C_VEL
LIN {X 0,Y 552.311,Z 402.769,A -85,B 0,C 180,E1 -3365.826,E2 -3365.826} C_VEL
LIN {X 0,Y 552.482,Z 397.791,A -85,B 0,C 180,E1 -3368.558,E2 -3368.558} C_VEL
LIN {X 0,Y 552.594,Z 392.961,A -85,B 0,C 180,E1 -3371.402,E2 -3371.402} C_VEL
LIN {X 0,Y 552.182,Z 389.788,A -85,B 0,C 180,E1 -3373.491,E2 -3373.491} C_VEL
LIN {X 0,Y 552.095,Z 389.215,A -85,B 0,C 180,E1 -3374.531,E2 -3374.531} C_VEL
LIN {X 0,Y 552.129,Z 389.209,A -85,B 0,C 180,E1 -3377.584,E2 -3377.584} C_VEL
LIN {X 0,Y 552.132,Z 389.208,A -85,B 0,C 180,E1 -3380.473,E2 -3380.473} C_VEL
LIN {X 0,Y 552.112,Z 389.212,A -85,B 0,C 180,E1 -3383.315,E2 -3383.315} C_VEL
LIN {X 0,Y 552.128,Z 389.204,A -85,B 0,C 180,E1 -3385.939,E2 -3385.939} C_VEL
LIN {X 0,Y 552.115,Z 389.21,A -85,B 0,C 180,E1 -3388.54,E2 -3388.54} C_VEL
LIN {X 0,Y 552.122,Z 389.206,A -85,B 0,C 180,E1 -3391.437,E2 -3391.437} C_VEL
LIN {X 0,Y 552.126,Z 389.207,A -85,B 0,C 180,E1 -3394.355,E2 -3394.355} C_VEL
LIN {X 0,Y 552.106,Z 389.217,A -85,B 0,C 180,E1 -3396.758,E2 -3396.758} C_VEL
LIN {X 0,Y 552.116,Z 389.209,A -85,B 0,C 180,E1 -3399.119,E2 -3399.119} C_VEL
LIN {X 0,Y 552.126,Z 389.205,A -85,B 0,C 180,E1 -3401.444,E2 -3401.444} C_VEL
LIN {X 0,Y 552.115,Z 389.206,A -85,B 0,C 180,E1 -3403.737,E2 -3403.737} C_VEL
LIN {X 0,Y 552.132,Z 389.205,A -85,B 0,C 180,E1 -3406.004,E2 -3406.004} C_VEL
LIN {X 0,Y 552.156,Z 389.204,A -85,B 0,C 180,E1 -3408.993,E2 -3408.993} C_VEL
LIN {X 0,Y 552.155,Z 389.203,A -85,B 0,C 180,E1 -3411.951,E2 -3411.951} C_VEL
LIN {X 0,Y 552.226,Z 389.195,A -85,B 0,C 180,E1 -3414.889,E2 -3414.889} C_VEL
LIN {X 0,Y 552.218,Z 389.194,A -85,B 0,C 180,E1 -3417.811,E2 -3417.811} C_VEL
LIN {X 0,Y 552.238,Z 389.194,A -85,B 0,C 180,E1 -3420.729,E2 -3420.729} C_VEL
LIN {X 0,Y 552.203,Z 389.196,A -85,B 0,C 180,E1 -3422.918,E2 -3422.918} C_VEL
LIN {X 0,Y 552.195,Z 389.199,A -85,B 0,C 180,E1 -3425.844,E2 -3425.844} C_VEL
LIN {X 0,Y 552.157,Z 389.203,A -85,B 0,C 180,E1 -3428.785,E2 -3428.785} C_VEL
LIN {X 0,Y 552.155,Z 389.204,A -85,B 0,C 180,E1 -3431.75,E2 -3431.75} C_VEL
LIN {X 0,Y 552.129,Z 389.206,A -85,B 0,C 180,E1 -3434.748,E2 -3434.748} C_VEL
LIN {X 0,Y 552.108,Z 389.211,A -85,B 0,C 180,E1 -3437.788,E2 -3437.788} C_VEL
LIN {X 0,Y 552.124,Z 389.214,A -85,B 0,C 180,E1 -3440.101,E2 -3440.101} C_VEL
LIN {X 0,Y 552.089,Z 389.212,A -85,B 0,C 180,E1 -3442.451,E2 -3442.451} C_VEL
LIN {X 0,Y 552.149,Z 389.203,A -85,B 0,C 180,E1 -3445.351,E2 -3445.351} C_VEL
LIN {X 0,Y 552.12,Z 389.212,A -85,B 0,C 180,E1 -3448.097,E2 -3448.097} C_VEL
LIN {X 0,Y 552.106,Z 389.208,A -85,B 0,C 180,E1 -3450.619,E2 -3450.619} C_VEL
LIN {X 0,Y 552.122,Z 389.206,A -85,B 0,C 180,E1 -3453.185,E2 -3453.185} C_VEL
LIN {X 0,Y 552.116,Z 389.209,A -85,B 0,C 180,E1 -3453.8,E2 -3453.8} C_VEL
LIN {X 0,Y 551.482,Z 389.291,A -85,B 0,C 180,E1 -3454.408,E2 -3454.408} C_VEL
LIN {X 0,Y 548.656,Z 389.641,A -85,B 0,C 180,E1 -3455.396,E2 -3455.396} C_VEL
LIN {X 0,Y 546.231,Z 389.943,A -85,B 0,C 180,E1 -3456.192,E2 -3456.192} C_VEL
LIN {X 0,Y 545.16,Z 390.072,A -85,B 0,C 180,E1 -3456.805,E2 -3456.805} C_VEL
LIN {X 0,Y 545.058,Z 390.085,A -85,B 0,C 180,E1 -3457.013,E2 -3457.013} C_VEL
LIN {X 0,Y 545.086,Z 390.085,A -85,B 0,C 180,E1 -3460.14,E2 -3460.14} C_VEL
LIN {X 0,Y 545.079,Z 390.083,A -85,B 0,C 180,E1 -3463.106,E2 -3463.106} C_VEL
LIN {X 0,Y 545.059,Z 390.087,A -85,B 0,C 180,E1 -3466.224,E2 -3466.224} C_VEL
LIN {X 0,Y 545.095,Z 390.081,A -85,B 0,C 180,E1 -3468.888,E2 -3468.888} C_VEL
LIN {X 0,Y 545.048,Z 390.093,A -85,B 0,C 180,E1 -3471.763,E2 -3471.763} C_VEL
LIN {X 0,Y 545.058,Z 390.085,A -85,B 0,C 180,E1 -3474.534,E2 -3474.534} C_VEL
LIN {X 0,Y 545.078,Z 390.087,A -85,B 0,C 180,E1 -3477.213,E2 -3477.213} C_VEL
LIN {X 0,Y 545.061,Z 390.089,A -85,B 0,C 180,E1 -3479.811,E2 -3479.811} C_VEL
LIN {X 0,Y 545.091,Z 390.081,A -85,B 0,C 180,E1 -3482.345,E2 -3482.345} C_VEL
LIN {X 0,Y 545.114,Z 390.08,A -85,B 0,C 180,E1 -3484.821,E2 -3484.821} C_VEL
LIN {X 0,Y 545.041,Z 390.095,A -85,B 0,C 180,E1 -3487.243,E2 -3487.243} C_VEL
LIN {X 0,Y 545.116,Z 390.078,A -85,B 0,C 180,E1 -3490.415,E2 -3490.415} C_VEL
LIN {X 0,Y 545.07,Z 390.09,A -85,B 0,C 180,E1 -3493.521,E2 -3493.521} C_VEL
LIN {X 0,Y 545.091,Z 390.083,A -85,B 0,C 180,E1 -3495.82,E2 -3495.82} C_VEL
LIN {X 0,Y 545.115,Z 390.083,A -85,B 0,C 180,E1 -3498.85,E2 -3498.85} C_VEL
LIN {X 0,Y 545.127,Z 390.078,A -85,B 0,C 180,E1 -3501.847,E2 -3501.847} C_VEL
LIN {X 0,Y 545.205,Z 390.074,A -85,B 0,C 180,E1 -3504.823,E2 -3504.823} C_VEL
LIN {X 0,Y 545.196,Z 390.069,A -85,B 0,C 180,E1 -3507.784,E2 -3507.784} C_VEL
LIN {X 0,Y 545.21,Z 390.073,A -85,B 0,C 180,E1 -3510.739,E2 -3510.739} C_VEL
LIN {X 0,Y 545.169,Z 390.08,A -85,B 0,C 180,E1 -3512.956,E2 -3512.956} C_VEL
LIN {X 0,Y 545.178,Z 390.071,A -85,B 0,C 180,E1 -3515.919,E2 -3515.919} C_VEL
LIN {X 0,Y 545.119,Z 390.086,A -85,B 0,C 180,E1 -3518.9,E2 -3518.9} C_VEL
LIN {X 0,Y 545.132,Z 390.076,A -85,B 0,C 180,E1 -3521.904,E2 -3521.904} C_VEL
LIN {X 0,Y 545.082,Z 390.09,A -85,B 0,C 180,E1 -3524.944,E2 -3524.944} C_VEL
LIN {X 0,Y 545.076,Z 390.085,A -85,B 0,C 180,E1 -3528.026,E2 -3528.026} C_VEL
LIN {X 0,Y 545.092,Z 390.085,A -85,B 0,C 180,E1 -3530.372,E2 -3530.372} C_VEL
LIN {X 0,Y 545.088,Z 390.081,A -85,B 0,C 180,E1 -3533.559,E2 -3533.559} C_VEL
LIN {X 0,Y 545.085,Z 390.083,A -85,B 0,C 180,E1 -3536,E2 -3536} C_VEL
LIN {X 0,Y 545.087,Z 390.088,A -85,B 0,C 180,E1 -3538.749,E2 -3538.749} C_VEL
LIN {X 0,Y 545.074,Z 390.083,A -85,B 0,C 180,E1 -3541.682,E2 -3541.682} C_VEL
LIN {X 0,Y 545.077,Z 390.09,A -85,B 0,C 180,E1 -3544.563,E2 -3544.563} C_VEL
LIN {X 0,Y 545.037,Z 390.087,A -85,B 0,C 180,E1 -3547.304,E2 -3547.304} C_VEL
LIN {X 0,Y 545.088,Z 390.087,A -85,B 0,C 180,E1 -3550.14,E2 -3550.14} C_VEL
LIN {X 0,Y 545.083,Z 390.082,A -85,B 0,C 180,E1 -3553.106,E2 -3553.106} C_VEL
LIN {X 0,Y 545.051,Z 390.094,A -85,B 0,C 180,E1 -3556.225,E2 -3556.225} C_VEL
LIN {X 0,Y 545.092,Z 390.082,A -85,B 0,C 180,E1 -3558.887,E2 -3558.887} C_VEL
LIN {X 0,Y 545.049,Z 390.089,A -85,B 0,C 180,E1 -3561.763,E2 -3561.763} C_VEL
LIN {X 0,Y 545.06,Z 390.088,A -85,B 0,C 180,E1 -3564.534,E2 -3564.534} C_VEL
LIN {X 0,Y 545.076,Z 390.082,A -85,B 0,C 180,E1 -3567.213,E2 -3567.213} C_VEL
LIN {X 0,Y 545.097,Z 390.085,A -85,B 0,C 180,E1 -3569.813,E2 -3569.813} C_VEL
LIN {X 0,Y 545.092,Z 390.081,A -85,B 0,C 180,E1 -3572.826,E2 -3572.826} C_VEL
LIN {X 0,Y 545.047,Z 390.09,A -85,B 0,C 180,E1 -3575.631,E2 -3575.631} C_VEL
LIN {X 0,Y 545.06,Z 390.084,A -85,B 0,C 180,E1 -3578.837,E2 -3578.837} C_VEL
LIN {X 0,Y 545.079,Z 390.083,A -85,B 0,C 180,E1 -3581.196,E2 -3581.196} C_VEL
LIN {X 0,Y 545.072,Z 390.087,A -85,B 0,C 180,E1 -3583.522,E2 -3583.522} C_VEL
LIN {X 0,Y 545.091,Z 390.09,A -85,B 0,C 180,E1 -3585.82,E2 -3585.82} C_VEL
LIN {X 0,Y 545.113,Z 390.078,A -85,B 0,C 180,E1 -3588.85,E2 -3588.85} C_VEL
LIN {X 0,Y 545.127,Z 390.084,A -85,B 0,C 180,E1 -3591.847,E2 -3591.847} C_VEL
LIN {X 0,Y 545.202,Z 390.067,A -85,B 0,C 180,E1 -3594.823,E2 -3594.823} C_VEL
LIN {X 0,Y 545.191,Z 390.076,A -85,B 0,C 180,E1 -3597.784,E2 -3597.784} C_VEL
LIN {X 0,Y 545.21,Z 390.066,A -85,B 0,C 180,E1 -3600.739,E2 -3600.739} C_VEL
LIN {X 0,Y 545.171,Z 390.072,A -85,B 0,C 180,E1 -3602.956,E2 -3602.956} C_VEL
LIN {X 0,Y 545.168,Z 390.075,A -85,B 0,C 180,E1 -3605.92,E2 -3605.92} C_VEL
LIN {X 0,Y 545.118,Z 390.079,A -85,B 0,C 180,E1 -3608.9,E2 -3608.9} C_VEL
LIN {X 0,Y 545.132,Z 390.078,A -85,B 0,C 180,E1 -3611.905,E2 -3611.905} C_VEL
LIN {X 0,Y 545.083,Z 390.085,A -85,B 0,C 180,E1 -3614.944,E2 -3614.944} C_VEL
LIN {X 0,Y 545.08,Z 390.083,A -85,B 0,C 180,E1 -3618.026,E2 -3618.026} C_VEL
LIN {X 0,Y 545.093,Z 390.08,A -85,B 0,C 180,E1 -3620.373,E2 -3620.373} C_VEL
LIN {X 0,Y 545.089,Z 390.086,A -85,B 0,C 180,E1 -3623.559,E2 -3623.559} C_VEL
LIN {X 0,Y 545.078,Z 390.083,A -85,B 0,C 180,E1 -3626.001,E2 -3626.001} C_VEL
LIN {X 0,Y 545.087,Z 390.084,A -85,B 0,C 180,E1 -3628.749,E2 -3628.749} C_VEL
LIN {X 0,Y 545.077,Z 390.084,A -85,B 0,C 180,E1 -3631.683,E2 -3631.683} C_VEL
LIN {X 0,Y 545.081,Z 390.084,A -85,B 0,C 180,E1 -3634.564,E2 -3634.564} C_VEL
LIN {X 0,Y 545.04,Z 390.094,A -85,B 0,C 180,E1 -3637.304,E2 -3637.304} C_VEL
LIN {X 0,Y 545.075,Z 390.086,A -85,B 0,C 180,E1 -3640.142,E2 -3640.142} C_VEL
LIN {X 0,Y 545.063,Z 390.092,A -85,B 0,C 180,E1 -3642.697,E2 -3642.697} C_VEL
LIN {X 0,Y 545.063,Z 390.093,A -85,B 0,C 180,E1 -3645.167,E2 -3645.167} C_VEL
LIN {X 0,Y 545.076,Z 390.166,A -85,B 0,C 180,E1 -3645.873,E2 -3645.873} C_VEL
LIN {X 0,Y 545.611,Z 393.836,A -85,B 0,C 180,E1 -3648.34,E2 -3648.34} C_VEL
LIN {X 0,Y 545.551,Z 397.998,A -85,B 0,C 180,E1 -3650.859,E2 -3650.859} C_VEL
LIN {X 0,Y 545.308,Z 402.922,A -85,B 0,C 180,E1 -3653.641,E2 -3653.641} C_VEL
LIN {X 0,Y 545.2,Z 407.997,A -85,B 0,C 180,E1 -3656.338,E2 -3656.338} C_VEL
LIN {X 0,Y 545.09,Z 413.327,A -85,B 0,C 180,E1 -3658.954,E2 -3658.954} C_VEL
LIN {X 0,Y 545.024,Z 418.716,A -85,B 0,C 180,E1 -3661.504,E2 -3661.504} C_VEL
LIN {X 0,Y 544.947,Z 425.27,A -85,B 0,C 180,E1 -3664.525,E2 -3664.525} C_VEL
LIN {X 0,Y 544.872,Z 431.292,A -85,B 0,C 180,E1 -3667.235,E2 -3667.235} C_VEL
LIN {X 0,Y 544.823,Z 436.681,A -85,B 0,C 180,E1 -3669.617,E2 -3669.617} C_VEL
LIN {X 0,Y 544.75,Z 442.071,A -85,B 0,C 180,E1 -3671.963,E2 -3671.963} C_VEL
LIN {X 0,Y 544.713,Z 449.257,A -85,B 0,C 180,E1 -3675.046,E2 -3675.046} C_VEL
LIN {X 0,Y 544.646,Z 453.523,A -85,B 0,C 180,E1 -3676.854,E2 -3676.854} C_VEL
LIN {X 0,Y 546.113,Z 463.196,A -85,B 0,C 180,E1 -3677.103,E2 -3677.103} C_VEL
LIN {X 0,Y 546.015,Z 474.384,A -85,B 0,C 180,E1 -3677.455,E2 -3677.455} C_VEL
LIN {X 0,Y 545.82,Z 485.441,A -85,B 0,C 180,E1 -3677.922,E2 -3677.922} C_VEL
LIN {X 0,Y 545.634,Z 497.422,A -85,B 0,C 180,E1 -3678.584,E2 -3678.584} C_VEL
LIN {X 0,Y 545.416,Z 509.078,A -85,B 0,C 180,E1 -3679.419,E2 -3679.419} C_VEL
LIN {X 0,Y 545.227,Z 517.572,A -85,B 0,C 180,E1 -3680.166,E2 -3680.166} C_VEL
LIN {X 0,Y 545.062,Z 526.375,A -85,B 0,C 180,E1 -3681.099,E2 -3681.099} C_VEL
LIN {X 0,Y 544.896,Z 535.008,A -85,B 0,C 180,E1 -3682.217,E2 -3682.217} C_VEL
LIN {X 0,Y 544.76,Z 542.281,A -85,B 0,C 180,E1 -3683.407,E2 -3683.407} C_VEL
LIN {X 0,Y 544.738,Z 547.363,A -85,B 0,C 180,E1 -3684.447,E2 -3684.447} C_VEL
LIN {X 0,Y 544.66,Z 551.66,A -85,B 0,C 180,E1 -3685.56,E2 -3685.56} C_VEL
LIN {X 0,Y 544.669,Z 553.968,A -85,B 0,C 180,E1 -3686.301,E2 -3686.301} C_VEL
LIN {X 0,Y 544.65,Z 555.787,A -85,B 0,C 180,E1 -3687.041,E2 -3687.041} C_VEL
LIN {X 0,Y 544.546,Z 558.191,A -85,B 0,C 180,E1 -3688.521,E2 -3688.521} C_VEL
LIN {X 0,Y 544.542,Z 558.781,A -85,B 0,C 180,E1 -3689.26,E2 -3689.26} C_VEL
LIN {X 0,Y 544.542,Z 558.781,A -85,B 0,C 180,E1 -3690.739,E2 -3690.739} C_VEL
LIN {X 0,Y 544.546,Z 558.191,A -85,B 0,C 180,E1 -3691.479,E2 -3691.479} C_VEL
LIN {X 0,Y 544.65,Z 555.788,A -85,B 0,C 180,E1 -3692.958,E2 -3692.958} C_VEL
LIN {X 0,Y 544.683,Z 552.873,A -85,B 0,C 180,E1 -3694.069,E2 -3694.069} C_VEL
LIN {X 0,Y 544.653,Z 548.922,A -85,B 0,C 180,E1 -3695.182,E2 -3695.182} C_VEL
LIN {X 0,Y 544.723,Z 543.629,A -85,B 0,C 180,E1 -3696.334,E2 -3696.334} C_VEL
LIN {X 0,Y 544.836,Z 537.443,A -85,B 0,C 180,E1 -3697.411,E2 -3697.411} C_VEL
LIN {X 0,Y 545.006,Z 529.495,A -85,B 0,C 180,E1 -3698.528,E2 -3698.528} C_VEL
LIN {X 0,Y 545.141,Z 521.354,A -85,B 0,C 180,E1 -3699.461,E2 -3699.461} C_VEL
LIN {X 0,Y 545.372,Z 511.347,A -85,B 0,C 180,E1 -3700.393,E2 -3700.393} C_VEL
LIN {X 0,Y 545.54,Z 501.526,A -85,B 0,C 180,E1 -3701.142,E2 -3701.142} C_VEL
LIN {X 0,Y 545.693,Z 490.598,A -85,B 0,C 180,E1 -3701.816,E2 -3701.816} C_VEL
LIN {X 0,Y 545.989,Z 476.966,A -85,B 0,C 180,E1 -3702.451,E2 -3702.451} C_VEL
LIN {X 0,Y 546.128,Z 464.955,A -85,B 0,C 180,E1 -3702.849,E2 -3702.849} C_VEL
LIN {X 0,Y 545.835,Z 460.495,A -85,B 0,C 180,E1 -3702.974,E2 -3702.974} C_VEL
LIN {X 0,Y 544.65,Z 453.524,A -85,B 0,C 180,E1 -3703.145,E2 -3703.145} C_VEL
LIN {X 0,Y 544.691,Z 447.461,A -85,B 0,C 180,E1 -3705.721,E2 -3705.721} C_VEL
LIN {X 0,Y 544.75,Z 442.071,A -85,B 0,C 180,E1 -3708.037,E2 -3708.037} C_VEL
LIN {X 0,Y 544.822,Z 436.682,A -85,B 0,C 180,E1 -3710.382,E2 -3710.382} C_VEL
LIN {X 0,Y 544.871,Z 431.292,A -85,B 0,C 180,E1 -3712.765,E2 -3712.765} C_VEL
LIN {X 0,Y 544.946,Z 425.271,A -85,B 0,C 180,E1 -3715.475,E2 -3715.475} C_VEL
LIN {X 0,Y 545.024,Z 418.717,A -85,B 0,C 180,E1 -3718.496,E2 -3718.496} C_VEL
LIN {X 0,Y 545.089,Z 413.327,A -85,B 0,C 180,E1 -3721.046,E2 -3721.046} C_VEL
LIN {X 0,Y 545.204,Z 407.998,A -85,B 0,C 180,E1 -3723.661,E2 -3723.661} C_VEL
LIN {X 0,Y 545.306,Z 402.923,A -85,B 0,C 180,E1 -3726.359,E2 -3726.359} C_VEL
LIN {X 0,Y 545.545,Z 397.974,A -85,B 0,C 180,E1 -3729.141,E2 -3729.141} C_VEL
LIN {X 0,Y 545.561,Z 393.84,A -85,B 0,C 180,E1 -3731.654,E2 -3731.654} C_VEL
LIN {X 0,Y 545.074,Z 390.174,A -85,B 0,C 180,E1 -3734.126,E2 -3734.126} C_VEL
LIN {X 0,Y 545.076,Z 390.091,A -85,B 0,C 180,E1 -3736.893,E2 -3736.893} C_VEL
LIN {X 0,Y 545.09,Z 390.086,A -85,B 0,C 180,E1 -3739.525,E2 -3739.525} C_VEL
LIN {X 0,Y 545.049,Z 390.088,A -85,B 0,C 180,E1 -3741.863,E2 -3741.863} C_VEL
LIN {X 0,Y 545.062,Z 390.09,A -85,B 0,C 180,E1 -3744.533,E2 -3744.533} C_VEL
LIN {X 0,Y 545.078,Z 390.087,A -85,B 0,C 180,E1 -3747.212,E2 -3747.212} C_VEL
LIN {X 0,Y 545.098,Z 390.08,A -85,B 0,C 180,E1 -3749.812,E2 -3749.812} C_VEL
LIN {X 0,Y 545.093,Z 390.09,A -85,B 0,C 180,E1 -3752.825,E2 -3752.825} C_VEL
LIN {X 0,Y 545.047,Z 390.086,A -85,B 0,C 180,E1 -3755.63,E2 -3755.63} C_VEL
LIN {X 0,Y 545.061,Z 390.092,A -85,B 0,C 180,E1 -3758.836,E2 -3758.836} C_VEL
LIN {X 0,Y 545.078,Z 390.084,A -85,B 0,C 180,E1 -3761.195,E2 -3761.195} C_VEL
LIN {X 0,Y 545.071,Z 390.083,A -85,B 0,C 180,E1 -3763.521,E2 -3763.521} C_VEL
LIN {X 0,Y 545.091,Z 390.081,A -85,B 0,C 180,E1 -3765.819,E2 -3765.819} C_VEL
LIN {X 0,Y 545.112,Z 390.083,A -85,B 0,C 180,E1 -3768.849,E2 -3768.849} C_VEL
LIN {X 0,Y 545.125,Z 390.077,A -85,B 0,C 180,E1 -3771.847,E2 -3771.847} C_VEL
LIN {X 0,Y 545.201,Z 390.071,A -85,B 0,C 180,E1 -3774.822,E2 -3774.822} C_VEL
LIN {X 0,Y 545.19,Z 390.07,A -85,B 0,C 180,E1 -3777.783,E2 -3777.783} C_VEL
LIN {X 0,Y 545.208,Z 390.07,A -85,B 0,C 180,E1 -3780.738,E2 -3780.738} C_VEL
LIN {X 0,Y 545.169,Z 390.072,A -85,B 0,C 180,E1 -3782.955,E2 -3782.955} C_VEL
LIN {X 0,Y 545.167,Z 390.075,A -85,B 0,C 180,E1 -3785.919,E2 -3785.919} C_VEL
LIN {X 0,Y 545.116,Z 390.079,A -85,B 0,C 180,E1 -3788.9,E2 -3788.9} C_VEL
LIN {X 0,Y 545.128,Z 390.081,A -85,B 0,C 180,E1 -3791.904,E2 -3791.904} C_VEL
LIN {X 0,Y 545.078,Z 390.083,A -85,B 0,C 180,E1 -3794.943,E2 -3794.943} C_VEL
LIN {X 0,Y 545.076,Z 390.091,A -85,B 0,C 180,E1 -3798.025,E2 -3798.025} C_VEL
LIN {X 0,Y 545.088,Z 390.086,A -85,B 0,C 180,E1 -3800.372,E2 -3800.372} C_VEL
LIN {X 0,Y 545.084,Z 390.084,A -85,B 0,C 180,E1 -3803.559,E2 -3803.559} C_VEL
LIN {X 0,Y 545.081,Z 390.092,A -85,B 0,C 180,E1 -3806,E2 -3806} C_VEL
LIN {X 0,Y 545.085,Z 390.082,A -85,B 0,C 180,E1 -3808.749,E2 -3808.749} C_VEL
LIN {X 0,Y 545.071,Z 390.089,A -85,B 0,C 180,E1 -3811.683,E2 -3811.683} C_VEL
LIN {X 0,Y 545.078,Z 390.083,A -85,B 0,C 180,E1 -3814.563,E2 -3814.563} C_VEL
LIN {X 0,Y 545.058,Z 390.085,A -85,B 0,C 180,E1 -3817.013,E2 -3817.013} C_VEL
LIN {X 0,Y 544.353,Z 390.18,A -85,B 0,C 180,E1 -3817.63,E2 -3817.63} C_VEL
LIN {X 0,Y 541.499,Z 390.536,A -85,B 0,C 180,E1 -3818.631,E2 -3818.631} C_VEL
LIN {X 0,Y 539.121,Z 390.832,A -85,B 0,C 180,E1 -3819.437,E2 -3819.437} C_VEL
LIN {X 0,Y 538.116,Z 390.955,A -85,B 0,C 180,E1 -3820.059,E2 -3820.059} C_VEL
LIN {X 0,Y 538.04,Z 390.961,A -85,B 0,C 180,E1 -3820.269,E2 -3820.269} C_VEL
LIN {X 0,Y 538.025,Z 390.961,A -85,B 0,C 180,E1 -3822.989,E2 -3822.989} C_VEL
LIN {X 0,Y 538.023,Z 390.967,A -85,B 0,C 180,E1 -3825.925,E2 -3825.925} C_VEL
LIN {X 0,Y 538.072,Z 390.959,A -85,B 0,C 180,E1 -3829.249,E2 -3829.249} C_VEL
LIN {X 0,Y 537.988,Z 390.967,A -85,B 0,C 180,E1 -3832.123,E2 -3832.123} C_VEL
LIN {X 0,Y 538.015,Z 390.963,A -85,B 0,C 180,E1 -3834.918,E2 -3834.918} C_VEL
LIN {X 0,Y 538.027,Z 390.968,A -85,B 0,C 180,E1 -3837.619,E2 -3837.619} C_VEL
LIN {X 0,Y 538.013,Z 390.963,A -85,B 0,C 180,E1 -3840.239,E2 -3840.239} C_VEL
LIN {X 0,Y 538.066,Z 390.957,A -85,B 0,C 180,E1 -3842.797,E2 -3842.797} C_VEL
LIN {X 0,Y 538.045,Z 390.967,A -85,B 0,C 180,E1 -3845.293,E2 -3845.293} C_VEL
LIN {X 0,Y 538.011,Z 390.963,A -85,B 0,C 180,E1 -3848.042,E2 -3848.042} C_VEL
LIN {X 0,Y 538.034,Z 390.964,A -85,B 0,C 180,E1 -3850.94,E2 -3850.94} C_VEL
LIN {X 0,Y 538.021,Z 390.971,A -85,B 0,C 180,E1 -3853.299,E2 -3853.299} C_VEL
LIN {X 0,Y 538.06,Z 390.961,A -85,B 0,C 180,E1 -3855.631,E2 -3855.631} C_VEL
LIN {X 0,Y 538.074,Z 390.958,A -85,B 0,C 180,E1 -3858.702,E2 -3858.702} C_VEL
LIN {X 0,Y 538.084,Z 390.957,A -85,B 0,C 180,E1 -3861.74,E2 -3861.74} C_VEL
LIN {X 0,Y 538.163,Z 390.95,A -85,B 0,C 180,E1 -3864.755,E2 -3864.755} C_VEL
LIN {X 0,Y 538.168,Z 390.945,A -85,B 0,C 180,E1 -3867.755,E2 -3867.755} C_VEL
LIN {X 0,Y 538.18,Z 390.949,A -85,B 0,C 180,E1 -3870.748,E2 -3870.748} C_VEL
LIN {X 0,Y 538.136,Z 390.956,A -85,B 0,C 180,E1 -3872.995,E2 -3872.995} C_VEL
LIN {X 0,Y 538.132,Z 390.949,A -85,B 0,C 180,E1 -3875.997,E2 -3875.997} C_VEL
LIN {X 0,Y 538.069,Z 390.964,A -85,B 0,C 180,E1 -3879.018,E2 -3879.018} C_VEL
LIN {X 0,Y 538.08,Z 390.955,A -85,B 0,C 180,E1 -3882.063,E2 -3882.063} C_VEL
LIN {X 0,Y 538.042,Z 390.964,A -85,B 0,C 180,E1 -3885.144,E2 -3885.144} C_VEL
LIN {X 0,Y 538.029,Z 390.965,A -85,B 0,C 180,E1 -3888.27,E2 -3888.27} C_VEL
LIN {X 0,Y 538.036,Z 390.969,A -85,B 0,C 180,E1 -3890.651,E2 -3890.651} C_VEL
LIN {X 0,Y 538.021,Z 390.962,A -85,B 0,C 180,E1 -3893.887,E2 -3893.887} C_VEL
LIN {X 0,Y 538.047,Z 390.964,A -85,B 0,C 180,E1 -3896.366,E2 -3896.366} C_VEL
LIN {X 0,Y 538.028,Z 390.964,A -85,B 0,C 180,E1 -3898.934,E2 -3898.934} C_VEL
LIN {X 0,Y 538.024,Z 390.962,A -85,B 0,C 180,E1 -3901.89,E2 -3901.89} C_VEL
LIN {X 0,Y 538.027,Z 390.968,A -85,B 0,C 180,E1 -3904.621,E2 -3904.621} C_VEL
LIN {X 0,Y 538.006,Z 390.964,A -85,B 0,C 180,E1 -3907.171,E2 -3907.171} C_VEL
LIN {X 0,Y 538.049,Z 390.959,A -85,B 0,C 180,E1 -3909.794,E2 -3909.794} C_VEL
LIN {X 0,Y 538.02,Z 390.964,A -85,B 0,C 180,E1 -3912.785,E2 -3912.785} C_VEL
LIN {X 0,Y 538.027,Z 390.961,A -85,B 0,C 180,E1 -3915.141,E2 -3915.141} C_VEL
LIN {X 0,Y 538.036,Z 390.969,A -85,B 0,C 180,E1 -3918.228,E2 -3918.228} C_VEL
LIN {X 0,Y 538.011,Z 390.963,A -85,B 0,C 180,E1 -3921.17,E2 -3921.17} C_VEL
LIN {X 0,Y 538.024,Z 390.969,A -85,B 0,C 180,E1 -3924.083,E2 -3924.083} C_VEL
LIN {X 0,Y 538.026,Z 390.962,A -85,B 0,C 180,E1 -3926.728,E2 -3926.728} C_VEL
LIN {X 0,Y 538.033,Z 390.962,A -85,B 0,C 180,E1 -3929.554,E2 -3929.554} C_VEL
LIN {X 0,Y 538.042,Z 390.967,A -85,B 0,C 180,E1 -3931.951,E2 -3931.951} C_VEL
LIN {X 0,Y 538.066,Z 390.959,A -85,B 0,C 180,E1 -3934.467,E2 -3934.467} C_VEL
LIN {X 0,Y 538.018,Z 390.962,A -85,B 0,C 180,E1 -3936.929,E2 -3936.929} C_VEL
LIN {X 0,Y 538.074,Z 390.961,A -85,B 0,C 180,E1 -3940.148,E2 -3940.148} C_VEL
LIN {X 0,Y 538.023,Z 390.963,A -85,B 0,C 180,E1 -3943.299,E2 -3943.299} C_VEL
LIN {X 0,Y 538.059,Z 390.963,A -85,B 0,C 180,E1 -3945.631,E2 -3945.631} C_VEL
LIN {X 0,Y 538.072,Z 390.955,A -85,B 0,C 180,E1 -3948.702,E2 -3948.702} C_VEL
LIN {X 0,Y 538.083,Z 390.963,A -85,B 0,C 180,E1 -3951.74,E2 -3951.74} C_VEL
LIN {X 0,Y 538.159,Z 390.944,A -85,B 0,C 180,E1 -3954.755,E2 -3954.755} C_VEL
LIN {X 0,Y 538.163,Z 390.951,A -85,B 0,C 180,E1 -3957.755,E2 -3957.755} C_VEL
LIN {X 0,Y 538.18,Z 390.942,A -85,B 0,C 180,E1 -3960.749,E2 -3960.749} C_VEL
LIN {X 0,Y 538.137,Z 390.949,A -85,B 0,C 180,E1 -3962.995,E2 -3962.995} C_VEL
LIN {X 0,Y 538.121,Z 390.952,A -85,B 0,C 180,E1 -3965.998,E2 -3965.998} C_VEL
LIN {X 0,Y 538.069,Z 390.958,A -85,B 0,C 180,E1 -3969.018,E2 -3969.018} C_VEL
LIN {X 0,Y 538.08,Z 390.955,A -85,B 0,C 180,E1 -3972.063,E2 -3972.063} C_VEL
LIN {X 0,Y 538.042,Z 390.964,A -85,B 0,C 180,E1 -3975.144,E2 -3975.144} C_VEL
LIN {X 0,Y 538.032,Z 390.96,A -85,B 0,C 180,E1 -3978.271,E2 -3978.271} C_VEL
LIN {X 0,Y 538.037,Z 390.961,A -85,B 0,C 180,E1 -3980.652,E2 -3980.652} C_VEL
LIN {X 0,Y 538.022,Z 390.962,A -85,B 0,C 180,E1 -3983.888,E2 -3983.888} C_VEL
LIN {X 0,Y 538.04,Z 390.959,A -85,B 0,C 180,E1 -3986.367,E2 -3986.367} C_VEL
LIN {X 0,Y 538.029,Z 390.966,A -85,B 0,C 180,E1 -3988.934,E2 -3988.934} C_VEL
LIN {X 0,Y 538.026,Z 390.961,A -85,B 0,C 180,E1 -3991.891,E2 -3991.891} C_VEL
LIN {X 0,Y 538.031,Z 390.963,A -85,B 0,C 180,E1 -3994.621,E2 -3994.621} C_VEL
LIN {X 0,Y 538.008,Z 390.972,A -85,B 0,C 180,E1 -3997.171,E2 -3997.171} C_VEL
LIN {X 0,Y 538.029,Z 390.964,A -85,B 0,C 180,E1 -3999.797,E2 -3999.797} C_VEL
LIN {X 0,Y 538.019,Z 390.971,A -85,B 0,C 180,E1 -4002.786,E2 -4002.786} C_VEL
LIN {X 0,Y 538.033,Z 390.968,A -85,B 0,C 180,E1 -4005.141,E2 -4005.141} C_VEL
LIN {X 0,Y 538.163,Z 391.945,A -85,B 0,C 180,E1 -4006.201,E2 -4006.201} C_VEL
LIN {X 0,Y 538.628,Z 395.002,A -85,B 0,C 180,E1 -4008.284,E2 -4008.284} C_VEL
LIN {X 0,Y 538.511,Z 399.795,A -85,B 0,C 180,E1 -4011.213,E2 -4011.213} C_VEL
LIN {X 0,Y 538.299,Z 404.782,A -85,B 0,C 180,E1 -4014.044,E2 -4014.044} C_VEL
LIN {X 0,Y 538.172,Z 409.83,A -85,B 0,C 180,E1 -4016.738,E2 -4016.738} C_VEL
LIN {X 0,Y 538.045,Z 415.492,A -85,B 0,C 180,E1 -4019.554,E2 -4019.554} C_VEL
LIN {X 0,Y 537.96,Z 420.513,A -85,B 0,C 180,E1 -4021.946,E2 -4021.946} C_VEL
LIN {X 0,Y 537.887,Z 425.902,A -85,B 0,C 180,E1 -4024.458,E2 -4024.458} C_VEL
LIN {X 0,Y 537.799,Z 431.292,A -85,B 0,C 180,E1 -4026.919,E2 -4026.919} C_VEL
LIN {X 0,Y 537.759,Z 436.681,A -85,B 0,C 180,E1 -4029.338,E2 -4029.338} C_VEL
LIN {X 0,Y 537.676,Z 442.071,A -85,B 0,C 180,E1 -4031.717,E2 -4031.717} C_VEL
LIN {X 0,Y 537.618,Z 449.257,A -85,B 0,C 180,E1 -4034.844,E2 -4034.844} C_VEL
LIN {X 0,Y 537.588,Z 453.523,A -85,B 0,C 180,E1 -4036.679,E2 -4036.679} C_VEL
LIN {X 0,Y 539.205,Z 464.054,A -85,B 0,C 180,E1 -4036.959,E2 -4036.959} C_VEL
LIN {X 0,Y 539.079,Z 475.661,A -85,B 0,C 180,E1 -4037.339,E2 -4037.339} C_VEL
LIN {X 0,Y 538.864,Z 487.406,A -85,B 0,C 180,E1 -4037.86,E2 -4037.86} C_VEL
LIN {X 0,Y 538.609,Z 499.706,A -85,B 0,C 180,E1 -4038.586,E2 -4038.586} C_VEL
LIN {X 0,Y 538.41,Z 510.205,A -85,B 0,C 180,E1 -4039.375,E2 -4039.375} C_VEL
LIN {X 0,Y 538.136,Z 519.479,A -85,B 0,C 180,E1 -4040.225,E2 -4040.225} C_VEL
LIN {X 0,Y 537.979,Z 527.989,A -85,B 0,C 180,E1 -4041.17,E2 -4041.17} C_VEL
LIN {X 0,Y 537.817,Z 536.249,A -85,B 0,C 180,E1 -4042.302,E2 -4042.302} C_VEL
LIN {X 0,Y 537.697,Z 542.686,A -85,B 0,C 180,E1 -4043.397,E2 -4043.397} C_VEL
LIN {X 0,Y 537.673,Z 547.363,A -85,B 0,C 180,E1 -4044.374,E2 -4044.374} C_VEL
LIN {X 0,Y 537.557,Z 551.659,A -85,B 0,C 180,E1 -4045.501,E2 -4045.501} C_VEL
LIN {X 0,Y 537.591,Z 553.969,A -85,B 0,C 180,E1 -4046.252,E2 -4046.252} C_VEL
LIN {X 0,Y 537.551,Z 555.784,A -85,B 0,C 180,E1 -4047.002,E2 -4047.002} C_VEL
LIN {X 0,Y 537.452,Z 558.192,A -85,B 0,C 180,E1 -4048.501,E2 -4048.501} C_VEL
LIN {X 0,Y 537.442,Z 558.781,A -85,B 0,C 180,E1 -4049.251,E2 -4049.251} C_VEL
LIN {X 0,Y 537.442,Z 558.781,A -85,B 0,C 180,E1 -4050.749,E2 -4050.749} C_VEL
LIN {X 0,Y 537.452,Z 558.192,A -85,B 0,C 180,E1 -4051.498,E2 -4051.498} C_VEL
LIN {X 0,Y 537.551,Z 555.785,A -85,B 0,C 180,E1 -4052.998,E2 -4052.998} C_VEL
LIN {X 0,Y 537.603,Z 552.869,A -85,B 0,C 180,E1 -4054.123,E2 -4054.123} C_VEL
LIN {X 0,Y 537.586,Z 548.917,A -85,B 0,C 180,E1 -4055.25,E2 -4055.25} C_VEL
LIN {X 0,Y 537.638,Z 544.124,A -85,B 0,C 180,E1 -4056.319,E2 -4056.319} C_VEL
LIN {X 0,Y 537.754,Z 538.589,A -85,B 0,C 180,E1 -4057.321,E2 -4057.321} C_VEL
LIN {X 0,Y 537.883,Z 532.297,A -85,B 0,C 180,E1 -4058.263,E2 -4058.263} C_VEL
LIN {X 0,Y 538.052,Z 524.752,A -85,B 0,C 180,E1 -4059.207,E2 -4059.207} C_VEL
LIN {X 0,Y 538.231,Z 515.635,A -85,B 0,C 180,E1 -4060.153,E2 -4060.153} C_VEL
LIN {X 0,Y 538.533,Z 504.21,A -85,B 0,C 180,E1 -4061.098,E2 -4061.098} C_VEL
LIN {X 0,Y 538.657,Z 494.025,A -85,B 0,C 180,E1 -4061.772,E2 -4061.772} C_VEL
LIN {X 0,Y 538.924,Z 483.439,A -85,B 0,C 180,E1 -4062.33,E2 -4062.33} C_VEL
LIN {X 0,Y 539.101,Z 471.805,A -85,B 0,C 180,E1 -4062.804,E2 -4062.804} C_VEL
LIN {X 0,Y 539.065,Z 462.317,A -85,B 0,C 180,E1 -4063.092,E2 -4063.092} C_VEL
LIN {X 0,Y 537.594,Z 453.524,A -85,B 0,C 180,E1 -4063.321,E2 -4063.321} C_VEL
LIN {X 0,Y 537.626,Z 447.461,A -85,B 0,C 180,E1 -4065.933,E2 -4065.933} C_VEL
LIN {X 0,Y 537.733,Z 440.275,A -85,B 0,C 180,E1 -4069.071,E2 -4069.071} C_VEL
LIN {X 0,Y 537.805,Z 433.089,A -85,B 0,C 180,E1 -4072.269,E2 -4072.269} C_VEL
LIN {X 0,Y 537.858,Z 427.699,A -85,B 0,C 180,E1 -4074.716,E2 -4074.716} C_VEL
LIN {X 0,Y 537.935,Z 422.063,A -85,B 0,C 180,E1 -4077.326,E2 -4077.326} C_VEL
LIN {X 0,Y 538.029,Z 416.92,A -85,B 0,C 180,E1 -4079.76,E2 -4079.76} C_VEL
LIN {X 0,Y 538.133,Z 411.584,A -85,B 0,C 180,E1 -4082.374,E2 -4082.374} C_VEL
LIN {X 0,Y 538.24,Z 406.403,A -85,B 0,C 180,E1 -4085.065,E2 -4085.065} C_VEL
LIN {X 0,Y 538.428,Z 401.411,A -85,B 0,C 180,E1 -4087.841,E2 -4087.841} C_VEL
LIN {X 0,Y 538.603,Z 396.423,A -85,B 0,C 180,E1 -4090.815,E2 -4090.815} C_VEL
LIN {X 0,Y 538.349,Z 393.058,A -85,B 0,C 180,E1 -4093.024,E2 -4093.024} C_VEL
LIN {X 0,Y 538.114,Z 391.529,A -85,B 0,C 180,E1 -4094.083,E2 -4094.083} C_VEL
LIN {X 0,Y 538.03,Z 390.968,A -85,B 0,C 180,E1 -4095.14,E2 -4095.14} C_VEL
LIN {X 0,Y 538.039,Z 390.963,A -85,B 0,C 180,E1 -4098.227,E2 -4098.227} C_VEL
LIN {X 0,Y 538.013,Z 390.971,A -85,B 0,C 180,E1 -4101.169,E2 -4101.169} C_VEL
LIN {X 0,Y 538.027,Z 390.963,A -85,B 0,C 180,E1 -4104.083,E2 -4104.083} C_VEL
LIN {X 0,Y 538.028,Z 390.967,A -85,B 0,C 180,E1 -4106.727,E2 -4106.727} C_VEL
LIN {X 0,Y 538.034,Z 390.961,A -85,B 0,C 180,E1 -4109.553,E2 -4109.553} C_VEL
LIN {X 0,Y 538.043,Z 390.959,A -85,B 0,C 180,E1 -4111.95,E2 -4111.95} C_VEL
LIN {X 0,Y 538.067,Z 390.96,A -85,B 0,C 180,E1 -4114.467,E2 -4114.467} C_VEL
LIN {X 0,Y 538.018,Z 390.968,A -85,B 0,C 180,E1 -4116.928,E2 -4116.928} C_VEL
LIN {X 0,Y 538.074,Z 390.957,A -85,B 0,C 180,E1 -4120.147,E2 -4120.147} C_VEL
LIN {X 0,Y 538.022,Z 390.962,A -85,B 0,C 180,E1 -4123.299,E2 -4123.299} C_VEL
LIN {X 0,Y 538.059,Z 390.957,A -85,B 0,C 180,E1 -4125.63,E2 -4125.63} C_VEL
LIN {X 0,Y 538.071,Z 390.962,A -85,B 0,C 180,E1 -4128.701,E2 -4128.701} C_VEL
LIN {X 0,Y 538.082,Z 390.954,A -85,B 0,C 180,E1 -4131.739,E2 -4131.739} C_VEL
LIN {X 0,Y 538.158,Z 390.949,A -85,B 0,C 180,E1 -4134.755,E2 -4134.755} C_VEL
LIN {X 0,Y 538.162,Z 390.945,A -85,B 0,C 180,E1 -4137.754,E2 -4137.754} C_VEL
LIN {X 0,Y 538.178,Z 390.946,A -85,B 0,C 180,E1 -4140.748,E2 -4140.748} C_VEL
LIN {X 0,Y 538.135,Z 390.948,A -85,B 0,C 180,E1 -4142.994,E2 -4142.994} C_VEL
LIN {X 0,Y 538.119,Z 390.954,A -85,B 0,C 180,E1 -4145.997,E2 -4145.997} C_VEL
LIN {X 0,Y 538.066,Z 390.956,A -85,B 0,C 180,E1 -4149.017,E2 -4149.017} C_VEL
LIN {X 0,Y 538.076,Z 390.962,A -85,B 0,C 180,E1 -4152.062,E2 -4152.062} C_VEL
LIN {X 0,Y 538.038,Z 390.959,A -85,B 0,C 180,E1 -4155.143,E2 -4155.143} C_VEL
LIN {X 0,Y 538.028,Z 390.967,A -85,B 0,C 180,E1 -4158.27,E2 -4158.27} C_VEL
LIN {X 0,Y 538.032,Z 390.962,A -85,B 0,C 180,E1 -4160.651,E2 -4160.651} C_VEL
LIN {X 0,Y 538.016,Z 390.969,A -85,B 0,C 180,E1 -4163.887,E2 -4163.887} C_VEL
LIN {X 0,Y 538.043,Z 390.962,A -85,B 0,C 180,E1 -4166.366,E2 -4166.366} C_VEL
LIN {X 0,Y 538.049,Z 390.958,A -85,B 0,C 180,E1 -4168.939,E2 -4168.939} C_VEL
LIN {X 0,Y 538.021,Z 390.971,A -85,B 0,C 180,E1 -4171.89,E2 -4171.89} C_VEL
LIN {X 0,Y 538.027,Z 390.961,A -85,B 0,C 180,E1 -4174.621,E2 -4174.621} C_VEL
LIN {X 0,Y 538.001,Z 390.965,A -85,B 0,C 180,E1 -4177.171,E2 -4177.171} C_VEL
LIN {X 0,Y 538.04,Z 390.961,A -85,B 0,C 180,E1 -4180.269,E2 -4180.269} C_VEL
LIN {X 0,Y 537.389,Z 391.04,A -85,B 0,C 180,E1 -4180.895,E2 -4180.895} C_VEL
LIN {X 0,Y 534.529,Z 391.403,A -85,B 0,C 180,E1 -4181.909,E2 -4181.909} C_VEL
LIN {X 0,Y 532.096,Z 391.709,A -85,B 0,C 180,E1 -4182.726,E2 -4182.726} C_VEL
LIN {X 0,Y 531.044,Z 391.838,A -85,B 0,C 180,E1 -4183.357,E2 -4183.357} C_VEL
LIN {X 0,Y 530.956,Z 391.846,A -85,B 0,C 180,E1 -4183.57,E2 -4183.57} C_VEL
LIN {X 0,Y 530.961,Z 391.841,A -85,B 0,C 180,E1 -4186.506,E2 -4186.506} C_VEL
LIN {X 0,Y 531.02,Z 391.842,A -85,B 0,C 180,E1 -4189.572,E2 -4189.572} C_VEL
LIN {X 0,Y 530.964,Z 391.84,A -85,B 0,C 180,E1 -4192.577,E2 -4192.577} C_VEL
LIN {X 0,Y 530.998,Z 391.842,A -85,B 0,C 180,E1 -4195.312,E2 -4195.312} C_VEL
LIN {X 0,Y 530.978,Z 391.841,A -85,B 0,C 180,E1 -4198.033,E2 -4198.033} C_VEL
LIN {X 0,Y 530.984,Z 391.84,A -85,B 0,C 180,E1 -4200.874,E2 -4200.874} C_VEL
LIN {X 0,Y 531.007,Z 391.842,A -85,B 0,C 180,E1 -4203.257,E2 -4203.257} C_VEL
LIN {X 0,Y 530.992,Z 391.839,A -85,B 0,C 180,E1 -4205.958,E2 -4205.958} C_VEL
LIN {X 0,Y 530.995,Z 391.842,A -85,B 0,C 180,E1 -4209.062,E2 -4209.062} C_VEL
LIN {X 0,Y 531.012,Z 391.836,A -85,B 0,C 180,E1 -4212.278,E2 -4212.278} C_VEL
LIN {X 0,Y 531.015,Z 391.842,A -85,B 0,C 180,E1 -4215.436,E2 -4215.436} C_VEL
LIN {X 0,Y 531.034,Z 391.834,A -85,B 0,C 180,E1 -4218.55,E2 -4218.55} C_VEL
LIN {X 0,Y 531.054,Z 391.834,A -85,B 0,C 180,E1 -4221.63,E2 -4221.63} C_VEL
LIN {X 0,Y 531.122,Z 391.826,A -85,B 0,C 180,E1 -4224.686,E2 -4224.686} C_VEL
LIN {X 0,Y 531.139,Z 391.821,A -85,B 0,C 180,E1 -4227.725,E2 -4227.725} C_VEL
LIN {X 0,Y 531.15,Z 391.825,A -85,B 0,C 180,E1 -4230.758,E2 -4230.758} C_VEL
LIN {X 0,Y 531.102,Z 391.832,A -85,B 0,C 180,E1 -4233.034,E2 -4233.034} C_VEL
LIN {X 0,Y 531.09,Z 391.827,A -85,B 0,C 180,E1 -4236.077,E2 -4236.077} C_VEL
LIN {X 0,Y 531.029,Z 391.839,A -85,B 0,C 180,E1 -4239.138,E2 -4239.138} C_VEL
LIN {X 0,Y 531.038,Z 391.834,A -85,B 0,C 180,E1 -4242.225,E2 -4242.225} C_VEL
LIN {X 0,Y 530.992,Z 391.84,A -85,B 0,C 180,E1 -4245.35,E2 -4245.35} C_VEL
LIN {X 0,Y 530.988,Z 391.845,A -85,B 0,C 180,E1 -4248.521,E2 -4248.521} C_VEL
LIN {X 0,Y 530.996,Z 391.842,A -85,B 0,C 180,E1 -4250.938,E2 -4250.938} C_VEL
LIN {X 0,Y 530.977,Z 391.842,A -85,B 0,C 180,E1 -4254.224,E2 -4254.224} C_VEL
LIN {X 0,Y 531.008,Z 391.842,A -85,B 0,C 180,E1 -4256.743,E2 -4256.743} C_VEL
LIN {X 0,Y 530.979,Z 391.839,A -85,B 0,C 180,E1 -4259.323,E2 -4259.323} C_VEL
LIN {X 0,Y 530.976,Z 391.842,A -85,B 0,C 180,E1 -4262.103,E2 -4262.103} C_VEL
LIN {X 0,Y 530.984,Z 391.842,A -85,B 0,C 180,E1 -4264.854,E2 -4264.854} C_VEL
LIN {X 0,Y 530.963,Z 391.841,A -85,B 0,C 180,E1 -4267.507,E2 -4267.507} C_VEL
LIN {X 0,Y 531.022,Z 391.842,A -85,B 0,C 180,E1 -4270.429,E2 -4270.429} C_VEL
LIN {X 0,Y 530.962,Z 391.841,A -85,B 0,C 180,E1 -4273.494,E2 -4273.494} C_VEL
LIN {X 0,Y 530.954,Z 391.848,A -85,B 0,C 180,E1 -4276.505,E2 -4276.505} C_VEL
LIN {X 0,Y 530.984,Z 391.839,A -85,B 0,C 180,E1 -4278.976,E2 -4278.976} C_VEL
LIN {X 0,Y 530.954,Z 391.843,A -85,B 0,C 180,E1 -4281.53,E2 -4281.53} C_VEL
LIN {X 0,Y 530.977,Z 391.845,A -85,B 0,C 180,E1 -4284.382,E2 -4284.382} C_VEL
LIN {X 0,Y 530.967,Z 391.84,A -85,B 0,C 180,E1 -4287.134,E2 -4287.134} C_VEL
LIN {X 0,Y 530.981,Z 391.843,A -85,B 0,C 180,E1 -4289.804,E2 -4289.804} C_VEL
LIN {X 0,Y 531.011,Z 391.838,A -85,B 0,C 180,E1 -4292.467,E2 -4292.467} C_VEL
LIN {X 0,Y 531.001,Z 391.836,A -85,B 0,C 180,E1 -4294.943,E2 -4294.943} C_VEL
LIN {X 0,Y 530.966,Z 391.845,A -85,B 0,C 180,E1 -4298.247,E2 -4298.247} C_VEL
LIN {X 0,Y 530.992,Z 391.837,A -85,B 0,C 180,E1 -4300.678,E2 -4300.678} C_VEL
LIN {X 0,Y 530.988,Z 391.838,A -85,B 0,C 180,E1 -4303.072,E2 -4303.072} C_VEL
LIN {X 0,Y 531.014,Z 391.838,A -85,B 0,C 180,E1 -4305.436,E2 -4305.436} C_VEL
LIN {X 0,Y 531.032,Z 391.833,A -85,B 0,C 180,E1 -4308.55,E2 -4308.55} C_VEL
LIN {X 0,Y 531.053,Z 391.837,A -85,B 0,C 180,E1 -4311.63,E2 -4311.63} C_VEL
LIN {X 0,Y 531.118,Z 391.821,A -85,B 0,C 180,E1 -4314.686,E2 -4314.686} C_VEL
LIN {X 0,Y 531.135,Z 391.827,A -85,B 0,C 180,E1 -4317.725,E2 -4317.725} C_VEL
LIN {X 0,Y 531.15,Z 391.817,A -85,B 0,C 180,E1 -4320.759,E2 -4320.759} C_VEL
LIN {X 0,Y 531.104,Z 391.825,A -85,B 0,C 180,E1 -4323.035,E2 -4323.035} C_VEL
LIN {X 0,Y 531.081,Z 391.828,A -85,B 0,C 180,E1 -4326.078,E2 -4326.078} C_VEL
LIN {X 0,Y 531.029,Z 391.837,A -85,B 0,C 180,E1 -4329.139,E2 -4329.139} C_VEL
LIN {X 0,Y 531.038,Z 391.832,A -85,B 0,C 180,E1 -4332.225,E2 -4332.225} C_VEL
LIN {X 0,Y 530.993,Z 391.846,A -85,B 0,C 180,E1 -4335.35,E2 -4335.35} C_VEL
LIN {X 0,Y 530.99,Z 391.838,A -85,B 0,C 180,E1 -4338.522,E2 -4338.522} C_VEL
LIN {X 0,Y 530.997,Z 391.84,A -85,B 0,C 180,E1 -4340.938,E2 -4340.938} C_VEL
LIN {X 0,Y 530.978,Z 391.839,A -85,B 0,C 180,E1 -4344.225,E2 -4344.225} C_VEL
LIN {X 0,Y 531.003,Z 391.838,A -85,B 0,C 180,E1 -4346.744,E2 -4346.744} C_VEL
LIN {X 0,Y 530.98,Z 391.845,A -85,B 0,C 180,E1 -4349.323,E2 -4349.323} C_VEL
LIN {X 0,Y 530.979,Z 391.839,A -85,B 0,C 180,E1 -4352.103,E2 -4352.103} C_VEL
LIN {X 0,Y 530.988,Z 391.843,A -85,B 0,C 180,E1 -4354.855,E2 -4354.855} C_VEL
LIN {X 0,Y 530.966,Z 391.845,A -85,B 0,C 180,E1 -4357.508,E2 -4357.508} C_VEL
LIN {X 0,Y 530.985,Z 391.843,A -85,B 0,C 180,E1 -4360.433,E2 -4360.433} C_VEL
LIN {X 0,Y 530.967,Z 391.848,A -85,B 0,C 180,E1 -4363.282,E2 -4363.282} C_VEL
LIN {X 0,Y 530.989,Z 391.845,A -85,B 0,C 180,E1 -4364.547,E2 -4364.547} C_VEL
LIN {X 0,Y 531.06,Z 392.405,A -85,B 0,C 180,E1 -4365.613,E2 -4365.613} C_VEL
LIN {X 0,Y 531.531,Z 395.489,A -85,B 0,C 180,E1 -4367.77,E2 -4367.77} C_VEL
LIN {X 0,Y 531.57,Z 399.086,A -85,B 0,C 180,E1 -4370.071,E2 -4370.071} C_VEL
LIN {X 0,Y 531.385,Z 403.227,A -85,B 0,C 180,E1 -4372.527,E2 -4372.527} C_VEL
LIN {X 0,Y 531.199,Z 408.22,A -85,B 0,C 180,E1 -4375.326,E2 -4375.326} C_VEL
LIN {X 0,Y 531.097,Z 413.417,A -85,B 0,C 180,E1 -4378.041,E2 -4378.041} C_VEL
LIN {X 0,Y 530.968,Z 419.134,A -85,B 0,C 180,E1 -4380.879,E2 -4380.879} C_VEL
LIN {X 0,Y 530.85,Z 425.902,A -85,B 0,C 180,E1 -4384.095,E2 -4384.095} C_VEL
LIN {X 0,Y 530.742,Z 431.292,A -85,B 0,C 180,E1 -4386.594,E2 -4386.594} C_VEL
LIN {X 0,Y 530.715,Z 436.681,A -85,B 0,C 180,E1 -4389.05,E2 -4389.05} C_VEL
LIN {X 0,Y 530.605,Z 442.071,A -85,B 0,C 180,E1 -4391.465,E2 -4391.465} C_VEL
LIN {X 0,Y 530.54,Z 447.46,A -85,B 0,C 180,E1 -4393.848,E2 -4393.848} C_VEL
LIN {X 0,Y 530.518,Z 453.299,A -85,B 0,C 180,E1 -4396.4,E2 -4396.4} C_VEL
LIN {X 0,Y 530.493,Z 453.523,A -85,B 0,C 180,E1 -4396.497,E2 -4396.497} C_VEL
LIN {X 0,Y 532.299,Z 464.911,A -85,B 0,C 180,E1 -4396.811,E2 -4396.811} C_VEL
LIN {X 0,Y 532.131,Z 476.937,A -85,B 0,C 180,E1 -4397.219,E2 -4397.219} C_VEL
LIN {X 0,Y 531.884,Z 489.198,A -85,B 0,C 180,E1 -4397.795,E2 -4397.795} C_VEL
LIN {X 0,Y 531.644,Z 499.906,A -85,B 0,C 180,E1 -4398.448,E2 -4398.448} C_VEL
LIN {X 0,Y 531.376,Z 510.199,A -85,B 0,C 180,E1 -4399.233,E2 -4399.233} C_VEL
LIN {X 0,Y 531.116,Z 519.474,A -85,B 0,C 180,E1 -4400.095,E2 -4400.095} C_VEL
LIN {X 0,Y 530.94,Z 527.986,A -85,B 0,C 180,E1 -4401.052,E2 -4401.052} C_VEL
LIN {X 0,Y 530.758,Z 536.25,A -85,B 0,C 180,E1 -4402.199,E2 -4402.199} C_VEL
LIN {X 0,Y 530.596,Z 543.246,A -85,B 0,C 180,E1 -4403.421,E2 -4403.421} C_VEL
LIN {X 0,Y 530.523,Z 548.912,A -85,B 0,C 180,E1 -4404.679,E2 -4404.679} C_VEL
LIN {X 0,Y 530.522,Z 552.864,A -85,B 0,C 180,E1 -4405.822,E2 -4405.822} C_VEL
LIN {X 0,Y 530.457,Z 555.782,A -85,B 0,C 180,E1 -4406.962,E2 -4406.962} C_VEL
LIN {X 0,Y 530.361,Z 558.193,A -85,B 0,C 180,E1 -4408.481,E2 -4408.481} C_VEL
LIN {X 0,Y 530.344,Z 558.781,A -85,B 0,C 180,E1 -4409.241,E2 -4409.241} C_VEL
LIN {X 0,Y 530.344,Z 558.781,A -85,B 0,C 180,E1 -4410.759,E2 -4410.759} C_VEL
LIN {X 0,Y 530.361,Z 558.193,A -85,B 0,C 180,E1 -4411.518,E2 -4411.518} C_VEL
LIN {X 0,Y 530.457,Z 555.783,A -85,B 0,C 180,E1 -4413.038,E2 -4413.038} C_VEL
LIN {X 0,Y 530.522,Z 552.865,A -85,B 0,C 180,E1 -4414.178,E2 -4414.178} C_VEL
LIN {X 0,Y 530.523,Z 548.913,A -85,B 0,C 180,E1 -4415.32,E2 -4415.32} C_VEL
LIN {X 0,Y 530.593,Z 543.263,A -85,B 0,C 180,E1 -4416.575,E2 -4416.575} C_VEL
LIN {X 0,Y 530.758,Z 536.252,A -85,B 0,C 180,E1 -4417.8,E2 -4417.8} C_VEL
LIN {X 0,Y 530.94,Z 527.989,A -85,B 0,C 180,E1 -4418.947,E2 -4418.947} C_VEL
LIN {X 0,Y 531.115,Z 519.477,A -85,B 0,C 180,E1 -4419.905,E2 -4419.905} C_VEL
LIN {X 0,Y 531.375,Z 510.202,A -85,B 0,C 180,E1 -4420.767,E2 -4420.767} C_VEL
LIN {X 0,Y 531.64,Z 499.99,A -85,B 0,C 180,E1 -4421.546,E2 -4421.546} C_VEL
LIN {X 0,Y 531.858,Z 489.204,A -85,B 0,C 180,E1 -4422.206,E2 -4422.206} C_VEL
LIN {X 0,Y 532.126,Z 476.946,A -85,B 0,C 180,E1 -4422.781,E2 -4422.781} C_VEL
LIN {X 0,Y 532.298,Z 464.923,A -85,B 0,C 180,E1 -4423.189,E2 -4423.189} C_VEL
LIN {X 0,Y 530.499,Z 453.524,A -85,B 0,C 180,E1 -4423.503,E2 -4423.503} C_VEL
LIN {X 0,Y 530.54,Z 449.257,A -85,B 0,C 180,E1 -4425.363,E2 -4425.363} C_VEL
LIN {X 0,Y 530.597,Z 443.868,A -85,B 0,C 180,E1 -4427.736,E2 -4427.736} C_VEL
LIN {X 0,Y 530.702,Z 438.478,A -85,B 0,C 180,E1 -4430.139,E2 -4430.139} C_VEL
LIN {X 0,Y 530.745,Z 433.089,A -85,B 0,C 180,E1 -4432.582,E2 -4432.582} C_VEL
LIN {X 0,Y 530.845,Z 426.115,A -85,B 0,C 180,E1 -4435.806,E2 -4435.806} C_VEL
LIN {X 0,Y 530.924,Z 420.513,A -85,B 0,C 180,E1 -4438.459,E2 -4438.459} C_VEL
LIN {X 0,Y 531.024,Z 415.174,A -85,B 0,C 180,E1 -4441.074,E2 -4441.074} C_VEL
LIN {X 0,Y 531.174,Z 409.91,A -85,B 0,C 180,E1 -4443.758,E2 -4443.758} C_VEL
LIN {X 0,Y 531.303,Z 404.869,A -85,B 0,C 180,E1 -4446.53,E2 -4446.53} C_VEL
LIN {X 0,Y 531.495,Z 401.057,A -85,B 0,C 180,E1 -4448.724,E2 -4448.724} C_VEL
LIN {X 0,Y 531.609,Z 396.771,A -85,B 0,C 180,E1 -4451.376,E2 -4451.376} C_VEL
LIN {X 0,Y 531.246,Z 393.693,A -85,B 0,C 180,E1 -4453.465,E2 -4453.465} C_VEL
LIN {X 0,Y 531.042,Z 392.177,A -85,B 0,C 180,E1 -4454.54,E2 -4454.54} C_VEL
LIN {X 0,Y 530.963,Z 391.847,A -85,B 0,C 180,E1 -4456.505,E2 -4456.505} C_VEL
LIN {X 0,Y 530.987,Z 391.847,A -85,B 0,C 180,E1 -4458.975,E2 -4458.975} C_VEL
LIN {X 0,Y 530.957,Z 391.846,A -85,B 0,C 180,E1 -4461.529,E2 -4461.529} C_VEL
LIN {X 0,Y 530.979,Z 391.843,A -85,B 0,C 180,E1 -4464.381,E2 -4464.381} C_VEL
LIN {X 0,Y 530.969,Z 391.846,A -85,B 0,C 180,E1 -4467.133,E2 -4467.133} C_VEL
LIN {X 0,Y 530.982,Z 391.838,A -85,B 0,C 180,E1 -4469.803,E2 -4469.803} C_VEL
LIN {X 0,Y 531.012,Z 391.839,A -85,B 0,C 180,E1 -4472.466,E2 -4472.466} C_VEL
LIN {X 0,Y 531.001,Z 391.843,A -85,B 0,C 180,E1 -4474.942,E2 -4474.942} C_VEL
LIN {X 0,Y 530.966,Z 391.843,A -85,B 0,C 180,E1 -4478.246,E2 -4478.246} C_VEL
LIN {X 0,Y 530.993,Z 391.846,A -85,B 0,C 180,E1 -4480.677,E2 -4480.677} C_VEL
LIN {X 0,Y 530.987,Z 391.841,A -85,B 0,C 180,E1 -4483.071,E2 -4483.071} C_VEL
LIN {X 0,Y 531.014,Z 391.835,A -85,B 0,C 180,E1 -4485.435,E2 -4485.435} C_VEL
LIN {X 0,Y 531.031,Z 391.842,A -85,B 0,C 180,E1 -4488.549,E2 -4488.549} C_VEL
LIN {X 0,Y 531.051,Z 391.83,A -85,B 0,C 180,E1 -4491.629,E2 -4491.629} C_VEL
LIN {X 0,Y 531.117,Z 391.827,A -85,B 0,C 180,E1 -4494.685,E2 -4494.685} C_VEL
LIN {X 0,Y 531.134,Z 391.82,A -85,B 0,C 180,E1 -4497.725,E2 -4497.725} C_VEL
LIN {X 0,Y 531.148,Z 391.821,A -85,B 0,C 180,E1 -4500.758,E2 -4500.758} C_VEL
LIN {X 0,Y 531.102,Z 391.824,A -85,B 0,C 180,E1 -4503.034,E2 -4503.034} C_VEL
LIN {X 0,Y 531.078,Z 391.832,A -85,B 0,C 180,E1 -4506.077,E2 -4506.077} C_VEL
LIN {X 0,Y 531.026,Z 391.833,A -85,B 0,C 180,E1 -4509.138,E2 -4509.138} C_VEL
LIN {X 0,Y 531.034,Z 391.841,A -85,B 0,C 180,E1 -4512.225,E2 -4512.225} C_VEL
LIN {X 0,Y 530.989,Z 391.838,A -85,B 0,C 180,E1 -4515.349,E2 -4515.349} C_VEL
LIN {X 0,Y 531.009,Z 391.838,A -85,B 0,C 180,E1 -4517.722,E2 -4517.722} C_VEL
LIN {X 0,Y 530.992,Z 391.837,A -85,B 0,C 180,E1 -4520.938,E2 -4520.938} C_VEL
LIN {X 0,Y 530.972,Z 391.846,A -85,B 0,C 180,E1 -4524.224,E2 -4524.224} C_VEL
LIN {X 0,Y 531.005,Z 391.836,A -85,B 0,C 180,E1 -4526.743,E2 -4526.743} C_VEL
LIN {X 0,Y 530.993,Z 391.838,A -85,B 0,C 180,E1 -4529.321,E2 -4529.321} C_VEL
LIN {X 0,Y 530.973,Z 391.845,A -85,B 0,C 180,E1 -4532.103,E2 -4532.103} C_VEL
LIN {X 0,Y 530.984,Z 391.838,A -85,B 0,C 180,E1 -4534.855,E2 -4534.855} C_VEL
LIN {X 0,Y 530.959,Z 391.846,A -85,B 0,C 180,E1 -4537.508,E2 -4537.508} C_VEL
LIN {X 0,Y 531.001,Z 391.837,A -85,B 0,C 180,E1 -4540.43,E2 -4540.43} C_VEL
LIN {X 0,Y 530.959,Z 391.847,A -85,B 0,C 180,E1 -4543.495,E2 -4543.495} C_VEL
LIN {X 0,Y 530.956,Z 391.846,A -85,B 0,C 180,E1 -4543.57,E2 -4543.57} C_VEL
LIN {X 0,Y 530.283,Z 391.928,A -85,B 0,C 180,E1 -4544.204,E2 -4544.204} C_VEL
LIN {X 0,Y 527.437,Z 392.283,A -85,B 0,C 180,E1 -4545.233,E2 -4545.233} C_VEL
LIN {X 0,Y 525.035,Z 392.583,A -85,B 0,C 180,E1 -4546.061,E2 -4546.061} C_VEL
LIN {X 0,Y 524.002,Z 392.708,A -85,B 0,C 180,E1 -4546.701,E2 -4546.701} C_VEL
LIN {X 0,Y 523.917,Z 392.719,A -85,B 0,C 180,E1 -4546.917,E2 -4546.917} C_VEL
LIN {X 0,Y 523.972,Z 392.716,A -85,B 0,C 180,E1 -4549.924,E2 -4549.924} C_VEL
LIN {X 0,Y 523.907,Z 392.72,A -85,B 0,C 180,E1 -4552.869,E2 -4552.869} C_VEL
LIN {X 0,Y 523.94,Z 392.722,A -85,B 0,C 180,E1 -4555.711,E2 -4555.711} C_VEL
LIN {X 0,Y 523.926,Z 392.717,A -85,B 0,C 180,E1 -4558.457,E2 -4558.457} C_VEL
LIN {X 0,Y 523.935,Z 392.72,A -85,B 0,C 180,E1 -4561.126,E2 -4561.126} C_VEL
LIN {X 0,Y 523.981,Z 392.712,A -85,B 0,C 180,E1 -4563.98,E2 -4563.98} C_VEL
LIN {X 0,Y 523.932,Z 392.717,A -85,B 0,C 180,E1 -4566.271,E2 -4566.271} C_VEL
LIN {X 0,Y 523.942,Z 392.717,A -85,B 0,C 180,E1 -4568.767,E2 -4568.767} C_VEL
LIN {X 0,Y 523.948,Z 392.723,A -85,B 0,C 180,E1 -4571.221,E2 -4571.221} C_VEL
LIN {X 0,Y 523.933,Z 392.722,A -85,B 0,C 180,E1 -4573.639,E2 -4573.639} C_VEL
LIN {X 0,Y 523.936,Z 392.718,A -85,B 0,C 180,E1 -4576.028,E2 -4576.028} C_VEL
LIN {X 0,Y 524.008,Z 392.708,A -85,B 0,C 180,E1 -4578.394,E2 -4578.394} C_VEL
LIN {X 0,Y 524.002,Z 392.713,A -85,B 0,C 180,E1 -4581.516,E2 -4581.516} C_VEL
LIN {X 0,Y 524.084,Z 392.702,A -85,B 0,C 180,E1 -4584.614,E2 -4584.614} C_VEL
LIN {X 0,Y 524.111,Z 392.697,A -85,B 0,C 180,E1 -4587.695,E2 -4587.695} C_VEL
LIN {X 0,Y 524.12,Z 392.701,A -85,B 0,C 180,E1 -4590.768,E2 -4590.768} C_VEL
LIN {X 0,Y 524.069,Z 392.708,A -85,B 0,C 180,E1 -4593.075,E2 -4593.075} C_VEL
LIN {X 0,Y 524.051,Z 392.704,A -85,B 0,C 180,E1 -4596.159,E2 -4596.159} C_VEL
LIN {X 0,Y 523.997,Z 392.714,A -85,B 0,C 180,E1 -4599.262,E2 -4599.262} C_VEL
LIN {X 0,Y 524,Z 392.709,A -85,B 0,C 180,E1 -4601.74,E2 -4601.74} C_VEL
LIN {X 0,Y 523.989,Z 392.716,A -85,B 0,C 180,E1 -4605.052,E2 -4605.052} C_VEL
LIN {X 0,Y 523.961,Z 392.715,A -85,B 0,C 180,E1 -4607.969,E2 -4607.969} C_VEL
LIN {X 0,Y 523.968,Z 392.717,A -85,B 0,C 180,E1 -4610.41,E2 -4610.41} C_VEL
LIN {X 0,Y 523.913,Z 392.724,A -85,B 0,C 180,E1 -4612.893,E2 -4612.893} C_VEL
LIN {X 0,Y 523.951,Z 392.714,A -85,B 0,C 180,E1 -4615.419,E2 -4615.419} C_VEL
LIN {X 0,Y 523.967,Z 392.714,A -85,B 0,C 180,E1 -4617.999,E2 -4617.999} C_VEL
LIN {X 0,Y 523.943,Z 392.719,A -85,B 0,C 180,E1 -4620.855,E2 -4620.855} C_VEL
LIN {X 0,Y 523.957,Z 392.714,A -85,B 0,C 180,E1 -4623.735,E2 -4623.735} C_VEL
LIN {X 0,Y 523.921,Z 392.727,A -85,B 0,C 180,E1 -4626.405,E2 -4626.405} C_VEL
LIN {X 0,Y 523.927,Z 392.718,A -85,B 0,C 180,E1 -4629.084,E2 -4629.084} C_VEL
LIN {X 0,Y 523.968,Z 392.712,A -85,B 0,C 180,E1 -4631.312,E2 -4631.312} C_VEL
LIN {X 0,Y 523.951,Z 392.718,A -85,B 0,C 180,E1 -4634.691,E2 -4634.691} C_VEL
LIN {X 0,Y 523.951,Z 392.718,A -85,B 0,C 180,E1 -4637.882,E2 -4637.882} C_VEL
LIN {X 0,Y 523.919,Z 392.719,A -85,B 0,C 180,E1 -4640.916,E2 -4640.916} C_VEL
LIN {X 0,Y 523.923,Z 392.722,A -85,B 0,C 180,E1 -4643.828,E2 -4643.828} C_VEL
LIN {X 0,Y 523.938,Z 392.718,A -85,B 0,C 180,E1 -4646.636,E2 -4646.636} C_VEL
LIN {X 0,Y 523.959,Z 392.714,A -85,B 0,C 180,E1 -4649.356,E2 -4649.356} C_VEL
LIN {X 0,Y 523.974,Z 392.717,A -85,B 0,C 180,E1 -4652.281,E2 -4652.281} C_VEL
LIN {X 0,Y 523.948,Z 392.716,A -85,B 0,C 180,E1 -4654.582,E2 -4654.582} C_VEL
LIN {X 0,Y 523.912,Z 392.719,A -85,B 0,C 180,E1 -4657.107,E2 -4657.107} C_VEL
LIN {X 0,Y 523.973,Z 392.72,A -85,B 0,C 180,E1 -4659.866,E2 -4659.866} C_VEL
LIN {X 0,Y 523.966,Z 392.712,A -85,B 0,C 180,E1 -4662.838,E2 -4662.838} C_VEL
LIN {X 0,Y 523.972,Z 392.713,A -85,B 0,C 180,E1 -4665.236,E2 -4665.236} C_VEL
LIN {X 0,Y 524.007,Z 392.709,A -85,B 0,C 180,E1 -4668.394,E2 -4668.394} C_VEL
LIN {X 0,Y 524.001,Z 392.714,A -85,B 0,C 180,E1 -4671.516,E2 -4671.516} C_VEL
LIN {X 0,Y 524.08,Z 392.698,A -85,B 0,C 180,E1 -4674.614,E2 -4674.614} C_VEL
LIN {X 0,Y 524.107,Z 392.703,A -85,B 0,C 180,E1 -4677.695,E2 -4677.695} C_VEL
LIN {X 0,Y 524.12,Z 392.693,A -85,B 0,C 180,E1 -4680.769,E2 -4680.769} C_VEL
LIN {X 0,Y 524.07,Z 392.702,A -85,B 0,C 180,E1 -4683.075,E2 -4683.075} C_VEL
LIN {X 0,Y 524.043,Z 392.704,A -85,B 0,C 180,E1 -4686.159,E2 -4686.159} C_VEL
LIN {X 0,Y 523.997,Z 392.714,A -85,B 0,C 180,E1 -4689.262,E2 -4689.262} C_VEL
LIN {X 0,Y 523.999,Z 392.713,A -85,B 0,C 180,E1 -4691.74,E2 -4691.74} C_VEL
LIN {X 0,Y 523.99,Z 392.714,A -85,B 0,C 180,E1 -4695.053,E2 -4695.053} C_VEL
LIN {X 0,Y 523.962,Z 392.714,A -85,B 0,C 180,E1 -4697.969,E2 -4697.969} C_VEL
LIN {X 0,Y 523.969,Z 392.712,A -85,B 0,C 180,E1 -4700.411,E2 -4700.411} C_VEL
LIN {X 0,Y 523.915,Z 392.723,A -85,B 0,C 180,E1 -4702.894,E2 -4702.894} C_VEL
LIN {X 0,Y 523.951,Z 392.72,A -85,B 0,C 180,E1 -4705.419,E2 -4705.419} C_VEL
LIN {X 0,Y 523.968,Z 392.712,A -85,B 0,C 180,E1 -4707.999,E2 -4707.999} C_VEL
LIN {X 0,Y 523.946,Z 392.72,A -85,B 0,C 180,E1 -4710.856,E2 -4710.856} C_VEL
LIN {X 0,Y 523.96,Z 392.714,A -85,B 0,C 180,E1 -4713.735,E2 -4713.735} C_VEL
LIN {X 0,Y 523.922,Z 392.721,A -85,B 0,C 180,E1 -4716.405,E2 -4716.405} C_VEL
LIN {X 0,Y 523.924,Z 392.727,A -85,B 0,C 180,E1 -4719.085,E2 -4719.085} C_VEL
LIN {X 0,Y 523.956,Z 392.718,A -85,B 0,C 180,E1 -4722.119,E2 -4722.119} C_VEL
LIN {X 0,Y 523.962,Z 392.721,A -85,B 0,C 180,E1 -4724.693,E2 -4724.693} C_VEL
LIN {X 0,Y 524.24,Z 394.751,A -85,B 0,C 180,E1 -4726.38,E2 -4726.38} C_VEL
LIN {X 0,Y 524.645,Z 397.987,A -85,B 0,C 180,E1 -4728.605,E2 -4728.605} C_VEL
LIN {X 0,Y 524.516,Z 401.799,A -85,B 0,C 180,E1 -4731,E2 -4731} C_VEL
LIN {X 0,Y 524.289,Z 406.698,A -85,B 0,C 180,E1 -4733.857,E2 -4733.857} C_VEL
LIN {X 0,Y 524.123,Z 411.742,A -85,B 0,C 180,E1 -4736.649,E2 -4736.649} C_VEL
LIN {X 0,Y 523.998,Z 417.008,A -85,B 0,C 180,E1 -4739.359,E2 -4739.359} C_VEL
LIN {X 0,Y 523.852,Z 422.958,A -85,B 0,C 180,E1 -4742.308,E2 -4742.308} C_VEL
LIN {X 0,Y 523.75,Z 427.699,A -85,B 0,C 180,E1 -4744.571,E2 -4744.571} C_VEL
LIN {X 0,Y 523.692,Z 433.088,A -85,B 0,C 180,E1 -4747.097,E2 -4747.097} C_VEL
LIN {X 0,Y 523.64,Z 439.337,A -85,B 0,C 180,E1 -4749.969,E2 -4749.969} C_VEL
LIN {X 0,Y 523.496,Z 445.664,A -85,B 0,C 180,E1 -4752.821,E2 -4752.821} C_VEL
LIN {X 0,Y 523.457,Z 452.85,A -85,B 0,C 180,E1 -4756.015,E2 -4756.015} C_VEL
LIN {X 0,Y 523.444,Z 453.523,A -85,B 0,C 180,E1 -4756.312,E2 -4756.312} C_VEL
LIN {X 0,Y 525.366,Z 465.769,A -85,B 0,C 180,E1 -4756.658,E2 -4756.658} C_VEL
LIN {X 0,Y 525.178,Z 478.16,A -85,B 0,C 180,E1 -4757.096,E2 -4757.096} C_VEL
LIN {X 0,Y 524.877,Z 491.107,A -85,B 0,C 180,E1 -4757.74,E2 -4757.74} C_VEL
LIN {X 0,Y 524.644,Z 501.498,A -85,B 0,C 180,E1 -4758.408,E2 -4758.408} C_VEL
LIN {X 0,Y 524.358,Z 511.324,A -85,B 0,C 180,E1 -4759.185,E2 -4759.185} C_VEL
LIN {X 0,Y 524.087,Z 521.356,A -85,B 0,C 180,E1 -4760.155,E2 -4760.155} C_VEL
LIN {X 0,Y 523.854,Z 530.917,A -85,B 0,C 180,E1 -4761.319,E2 -4761.319} C_VEL
LIN {X 0,Y 523.665,Z 537.428,A -85,B 0,C 180,E1 -4762.287,E2 -4762.287} C_VEL
LIN {X 0,Y 523.525,Z 543.664,A -85,B 0,C 180,E1 -4763.418,E2 -4763.418} C_VEL
LIN {X 0,Y 523.462,Z 548.907,A -85,B 0,C 180,E1 -4764.607,E2 -4764.607} C_VEL
LIN {X 0,Y 523.441,Z 552.861,A -85,B 0,C 180,E1 -4765.765,E2 -4765.765} C_VEL
LIN {X 0,Y 523.368,Z 555.779,A -85,B 0,C 180,E1 -4766.921,E2 -4766.921} C_VEL
LIN {X 0,Y 523.275,Z 558.194,A -85,B 0,C 180,E1 -4768.461,E2 -4768.461} C_VEL
LIN {X 0,Y 523.25,Z 558.781,A -85,B 0,C 180,E1 -4769.23,E2 -4769.23} C_VEL
LIN {X 0,Y 523.25,Z 558.781,A -85,B 0,C 180,E1 -4770.769,E2 -4770.769} C_VEL
LIN {X 0,Y 523.275,Z 558.194,A -85,B 0,C 180,E1 -4771.539,E2 -4771.539} C_VEL
LIN {X 0,Y 523.368,Z 555.78,A -85,B 0,C 180,E1 -4773.079,E2 -4773.079} C_VEL
LIN {X 0,Y 523.441,Z 552.862,A -85,B 0,C 180,E1 -4774.235,E2 -4774.235} C_VEL
LIN {X 0,Y 523.462,Z 548.909,A -85,B 0,C 180,E1 -4775.392,E2 -4775.392} C_VEL
LIN {X 0,Y 523.517,Z 543.704,A -85,B 0,C 180,E1 -4776.574,E2 -4776.574} C_VEL
LIN {X 0,Y 523.664,Z 537.43,A -85,B 0,C 180,E1 -4777.713,E2 -4777.713} C_VEL
LIN {X 0,Y 523.863,Z 529.5,A -85,B 0,C 180,E1 -4778.875,E2 -4778.875} C_VEL
LIN {X 0,Y 524.086,Z 521.359,A -85,B 0,C 180,E1 -4779.844,E2 -4779.844} C_VEL
LIN {X 0,Y 524.358,Z 511.328,A -85,B 0,C 180,E1 -4780.815,E2 -4780.815} C_VEL
LIN {X 0,Y 524.644,Z 501.502,A -85,B 0,C 180,E1 -4781.591,E2 -4781.591} C_VEL
LIN {X 0,Y 524.849,Z 491.343,A -85,B 0,C 180,E1 -4782.246,E2 -4782.246} C_VEL
LIN {X 0,Y 525.184,Z 478.168,A -85,B 0,C 180,E1 -4782.903,E2 -4782.903} C_VEL
LIN {X 0,Y 525.368,Z 465.781,A -85,B 0,C 180,E1 -4783.341,E2 -4783.341} C_VEL
LIN {X 0,Y 523.563,Z 454.523,A -85,B 0,C 180,E1 -4783.663,E2 -4783.663} C_VEL
LIN {X 0,Y 523.449,Z 453.524,A -85,B 0,C 180,E1 -4783.688,E2 -4783.688} C_VEL
LIN {X 0,Y 523.45,Z 449.257,A -85,B 0,C 180,E1 -4785.576,E2 -4785.576} C_VEL
LIN {X 0,Y 523.522,Z 443.868,A -85,B 0,C 180,E1 -4787.984,E2 -4787.984} C_VEL
LIN {X 0,Y 523.628,Z 438.478,A -85,B 0,C 180,E1 -4790.424,E2 -4790.424} C_VEL
LIN {X 0,Y 523.691,Z 433.089,A -85,B 0,C 180,E1 -4792.903,E2 -4792.903} C_VEL
LIN {X 0,Y 523.805,Z 426.535,A -85,B 0,C 180,E1 -4795.978,E2 -4795.978} C_VEL
LIN {X 0,Y 523.894,Z 420.526,A -85,B 0,C 180,E1 -4798.877,E2 -4798.877} C_VEL
LIN {X 0,Y 524.012,Z 415.252,A -85,B 0,C 180,E1 -4801.537,E2 -4801.537} C_VEL
LIN {X 0,Y 524.153,Z 410.039,A -85,B 0,C 180,E1 -4804.273,E2 -4804.273} C_VEL
LIN {X 0,Y 524.337,Z 404.994,A -85,B 0,C 180,E1 -4807.096,E2 -4807.096} C_VEL
LIN {X 0,Y 524.506,Z 401.731,A -85,B 0,C 180,E1 -4809.032,E2 -4809.032} C_VEL
LIN {X 0,Y 524.625,Z 397.973,A -85,B 0,C 180,E1 -4811.393,E2 -4811.393} C_VEL
LIN {X 0,Y 524.238,Z 394.741,A -85,B 0,C 180,E1 -4813.62,E2 -4813.62} C_VEL
LIN {X 0,Y 523.96,Z 392.72,A -85,B 0,C 180,E1 -4815.307,E2 -4815.307} C_VEL
LIN {X 0,Y 523.959,Z 392.72,A -85,B 0,C 180,E1 -4818.688,E2 -4818.688} C_VEL
LIN {X 0,Y 523.914,Z 392.721,A -85,B 0,C 180,E1 -4821.898,E2 -4821.898} C_VEL
LIN {X 0,Y 523.935,Z 392.725,A -85,B 0,C 180,E1 -4824.908,E2 -4824.908} C_VEL
LIN {X 0,Y 523.939,Z 392.716,A -85,B 0,C 180,E1 -4827.678,E2 -4827.678} C_VEL
LIN {X 0,Y 523.966,Z 392.719,A -85,B 0,C 180,E1 -4830.673,E2 -4830.673} C_VEL
LIN {X 0,Y 523.971,Z 392.712,A -85,B 0,C 180,E1 -4833.728,E2 -4833.728} C_VEL
LIN {X 0,Y 523.932,Z 392.719,A -85,B 0,C 180,E1 -4836.27,E2 -4836.27} C_VEL
LIN {X 0,Y 523.941,Z 392.724,A -85,B 0,C 180,E1 -4838.766,E2 -4838.766} C_VEL
LIN {X 0,Y 523.949,Z 392.716,A -85,B 0,C 180,E1 -4841.22,E2 -4841.22} C_VEL
LIN {X 0,Y 523.935,Z 392.716,A -85,B 0,C 180,E1 -4843.638,E2 -4843.638} C_VEL
LIN {X 0,Y 523.935,Z 392.718,A -85,B 0,C 180,E1 -4846.027,E2 -4846.027} C_VEL
LIN {X 0,Y 524.006,Z 392.714,A -85,B 0,C 180,E1 -4848.394,E2 -4848.394} C_VEL
LIN {X 0,Y 523.999,Z 392.708,A -85,B 0,C 180,E1 -4851.516,E2 -4851.516} C_VEL
LIN {X 0,Y 524.078,Z 392.705,A -85,B 0,C 180,E1 -4854.613,E2 -4854.613} C_VEL
LIN {X 0,Y 524.106,Z 392.695,A -85,B 0,C 180,E1 -4857.694,E2 -4857.694} C_VEL
LIN {X 0,Y 524.118,Z 392.697,A -85,B 0,C 180,E1 -4860.768,E2 -4860.768} C_VEL
LIN {X 0,Y 524.068,Z 392.7,A -85,B 0,C 180,E1 -4863.074,E2 -4863.074} C_VEL
LIN {X 0,Y 524.04,Z 392.71,A -85,B 0,C 180,E1 -4866.159,E2 -4866.159} C_VEL
LIN {X 0,Y 523.994,Z 392.709,A -85,B 0,C 180,E1 -4869.261,E2 -4869.261} C_VEL
LIN {X 0,Y 523.995,Z 392.711,A -85,B 0,C 180,E1 -4871.739,E2 -4871.739} C_VEL
LIN {X 0,Y 523.985,Z 392.71,A -85,B 0,C 180,E1 -4875.052,E2 -4875.052} C_VEL
LIN {X 0,Y 523.957,Z 392.72,A -85,B 0,C 180,E1 -4877.969,E2 -4877.969} C_VEL
LIN {X 0,Y 523.964,Z 392.717,A -85,B 0,C 180,E1 -4880.41,E2 -4880.41} C_VEL
LIN {X 0,Y 523.909,Z 392.72,A -85,B 0,C 180,E1 -4882.893,E2 -4882.893} C_VEL
LIN {X 0,Y 523.947,Z 392.716,A -85,B 0,C 180,E1 -4885.418,E2 -4885.418} C_VEL
LIN {X 0,Y 523.963,Z 392.721,A -85,B 0,C 180,E1 -4887.999,E2 -4887.999} C_VEL
LIN {X 0,Y 523.945,Z 392.715,A -85,B 0,C 180,E1 -4890.856,E2 -4890.856} C_VEL
LIN {X 0,Y 523.955,Z 392.721,A -85,B 0,C 180,E1 -4893.735,E2 -4893.735} C_VEL
LIN {X 0,Y 523.915,Z 392.72,A -85,B 0,C 180,E1 -4896.404,E2 -4896.404} C_VEL
LIN {X 0,Y 523.953,Z 392.715,A -85,B 0,C 180,E1 -4899.081,E2 -4899.081} C_VEL
LIN {X 0,Y 523.95,Z 392.718,A -85,B 0,C 180,E1 -4902.118,E2 -4902.118} C_VEL
LIN {X 0,Y 523.949,Z 392.718,A -85,B 0,C 180,E1 -4905.309,E2 -4905.309} C_VEL
LIN {X 0,Y 523.917,Z 392.719,A -85,B 0,C 180,E1 -4906.917,E2 -4906.917} C_VEL
LIN {X 0,Y 523.253,Z 392.809,A -85,B 0,C 180,E1 -4907.559,E2 -4907.559} C_VEL
LIN {X 0,Y 520.423,Z 393.16,A -85,B 0,C 180,E1 -4908.601,E2 -4908.601} C_VEL
LIN {X 0,Y 518.025,Z 393.459,A -85,B 0,C 180,E1 -4909.44,E2 -4909.44} C_VEL
LIN {X 0,Y 516.985,Z 393.585,A -85,B 0,C 180,E1 -4910.088,E2 -4910.088} C_VEL
LIN {X 0,Y 516.895,Z 393.594,A -85,B 0,C 180,E1 -4910.307,E2 -4910.307} C_VEL
LIN {X 0,Y 516.88,Z 393.601,A -85,B 0,C 180,E1 -4913.342,E2 -4913.342} C_VEL
LIN {X 0,Y 516.908,Z 393.593,A -85,B 0,C 180,E1 -4916.121,E2 -4916.121} C_VEL
LIN {X 0,Y 516.887,Z 393.596,A -85,B 0,C 180,E1 -4918.936,E2 -4918.936} C_VEL
LIN {X 0,Y 516.915,Z 393.598,A -85,B 0,C 180,E1 -4921.585,E2 -4921.585} C_VEL
LIN {X 0,Y 516.928,Z 393.589,A -85,B 0,C 180,E1 -4924.211,E2 -4924.211} C_VEL
LIN {X 0,Y 516.867,Z 393.598,A -85,B 0,C 180,E1 -4926.777,E2 -4926.777} C_VEL
LIN {X 0,Y 516.935,Z 393.592,A -85,B 0,C 180,E1 -4929.732,E2 -4929.732} C_VEL
LIN {X 0,Y 516.925,Z 393.592,A -85,B 0,C 180,E1 -4932.596,E2 -4932.596} C_VEL
LIN {X 0,Y 516.938,Z 393.596,A -85,B 0,C 180,E1 -4935.03,E2 -4935.03} C_VEL
LIN {X 0,Y 516.961,Z 393.586,A -85,B 0,C 180,E1 -4938.234,E2 -4938.234} C_VEL
LIN {X 0,Y 516.967,Z 393.591,A -85,B 0,C 180,E1 -4941.4,E2 -4941.4} C_VEL
LIN {X 0,Y 517.012,Z 393.582,A -85,B 0,C 180,E1 -4943.757,E2 -4943.757} C_VEL
LIN {X 0,Y 517.083,Z 393.573,A -85,B 0,C 180,E1 -4947.663,E2 -4947.663} C_VEL
LIN {X 0,Y 517.091,Z 393.576,A -85,B 0,C 180,E1 -4950.779,E2 -4950.779} C_VEL
LIN {X 0,Y 517.01,Z 393.587,A -85,B 0,C 180,E1 -4953.117,E2 -4953.117} C_VEL
LIN {X 0,Y 517.014,Z 393.582,A -85,B 0,C 180,E1 -4956.243,E2 -4956.243} C_VEL
LIN {X 0,Y 516.952,Z 393.591,A -85,B 0,C 180,E1 -4959.389,E2 -4959.389} C_VEL
LIN {X 0,Y 516.949,Z 393.588,A -85,B 0,C 180,E1 -4961.808,E2 -4961.808} C_VEL
LIN {X 0,Y 516.941,Z 393.593,A -85,B 0,C 180,E1 -4965.147,E2 -4965.147} C_VEL
LIN {X 0,Y 516.922,Z 393.594,A -85,B 0,C 180,E1 -4968.222,E2 -4968.222} C_VEL
LIN {X 0,Y 516.909,Z 393.6,A -85,B 0,C 180,E1 -4970.701,E2 -4970.701} C_VEL
LIN {X 0,Y 516.908,Z 393.593,A -85,B 0,C 180,E1 -4974.072,E2 -4974.072} C_VEL
LIN {X 0,Y 516.925,Z 393.598,A -85,B 0,C 180,E1 -4976.658,E2 -4976.658} C_VEL
LIN {X 0,Y 516.907,Z 393.592,A -85,B 0,C 180,E1 -4979.524,E2 -4979.524} C_VEL
LIN {X 0,Y 516.897,Z 393.602,A -85,B 0,C 180,E1 -4982.544,E2 -4982.544} C_VEL
LIN {X 0,Y 516.879,Z 393.595,A -85,B 0,C 180,E1 -4985.332,E2 -4985.332} C_VEL
LIN {X 0,Y 516.877,Z 393.598,A -85,B 0,C 180,E1 -4987.943,E2 -4987.943} C_VEL
LIN {X 0,Y 516.899,Z 393.596,A -85,B 0,C 180,E1 -4990.74,E2 -4990.74} C_VEL
LIN {X 0,Y 516.878,Z 393.598,A -85,B 0,C 180,E1 -4993.903,E2 -4993.903} C_VEL
LIN {X 0,Y 516.877,Z 393.602,A -85,B 0,C 180,E1 -4996.107,E2 -4996.107} C_VEL
LIN {X 0,Y 516.912,Z 393.598,A -85,B 0,C 180,E1 -4998.398,E2 -4998.398} C_VEL
LIN {X 0,Y 516.878,Z 393.595,A -85,B 0,C 180,E1 -5001.285,E2 -5001.285} C_VEL
LIN {X 0,Y 516.886,Z 393.603,A -85,B 0,C 180,E1 -5004.221,E2 -5004.221} C_VEL
LIN {X 0,Y 516.892,Z 393.593,A -85,B 0,C 180,E1 -5007.053,E2 -5007.053} C_VEL
LIN {X 0,Y 516.897,Z 393.598,A -85,B 0,C 180,E1 -5009.797,E2 -5009.797} C_VEL
LIN {X 0,Y 516.924,Z 393.593,A -85,B 0,C 180,E1 -5012.468,E2 -5012.468} C_VEL
LIN {X 0,Y 516.905,Z 393.592,A -85,B 0,C 180,E1 -5015.072,E2 -5015.072} C_VEL
LIN {X 0,Y 516.864,Z 393.601,A -85,B 0,C 180,E1 -5017.622,E2 -5017.622} C_VEL
LIN {X 0,Y 516.927,Z 393.595,A -85,B 0,C 180,E1 -5020.13,E2 -5020.13} C_VEL
LIN {X 0,Y 516.926,Z 393.59,A -85,B 0,C 180,E1 -5022.597,E2 -5022.597} C_VEL
LIN {X 0,Y 516.937,Z 393.588,A -85,B 0,C 180,E1 -5025.03,E2 -5025.03} C_VEL
LIN {X 0,Y 516.96,Z 393.588,A -85,B 0,C 180,E1 -5028.234,E2 -5028.234} C_VEL
LIN {X 0,Y 516.966,Z 393.588,A -85,B 0,C 180,E1 -5031.4,E2 -5031.4} C_VEL
LIN {X 0,Y 517.006,Z 393.588,A -85,B 0,C 180,E1 -5033.757,E2 -5033.757} C_VEL
LIN {X 0,Y 517.08,Z 393.579,A -85,B 0,C 180,E1 -5037.664,E2 -5037.664} C_VEL
LIN {X 0,Y 517.09,Z 393.569,A -85,B 0,C 180,E1 -5040.779,E2 -5040.779} C_VEL
LIN {X 0,Y 517.011,Z 393.582,A -85,B 0,C 180,E1 -5043.117,E2 -5043.117} C_VEL
LIN {X 0,Y 517.007,Z 393.58,A -85,B 0,C 180,E1 -5046.244,E2 -5046.244} C_VEL
LIN {X 0,Y 516.951,Z 393.594,A -85,B 0,C 180,E1 -5049.39,E2 -5049.39} C_VEL
LIN {X 0,Y 516.949,Z 393.59,A -85,B 0,C 180,E1 -5051.808,E2 -5051.808} C_VEL
LIN {X 0,Y 516.941,Z 393.593,A -85,B 0,C 180,E1 -5055.147,E2 -5055.147} C_VEL
LIN {X 0,Y 516.923,Z 393.59,A -85,B 0,C 180,E1 -5058.223,E2 -5058.223} C_VEL
LIN {X 0,Y 516.91,Z 393.593,A -85,B 0,C 180,E1 -5060.702,E2 -5060.702} C_VEL
LIN {X 0,Y 516.909,Z 393.592,A -85,B 0,C 180,E1 -5064.073,E2 -5064.073} C_VEL
LIN {X 0,Y 516.924,Z 393.591,A -85,B 0,C 180,E1 -5066.658,E2 -5066.658} C_VEL
LIN {X 0,Y 516.909,Z 393.595,A -85,B 0,C 180,E1 -5069.524,E2 -5069.524} C_VEL
LIN {X 0,Y 516.899,Z 393.594,A -85,B 0,C 180,E1 -5072.545,E2 -5072.545} C_VEL
LIN {X 0,Y 516.882,Z 393.602,A -85,B 0,C 180,E1 -5075.333,E2 -5075.333} C_VEL
LIN {X 0,Y 516.881,Z 393.598,A -85,B 0,C 180,E1 -5077.944,E2 -5077.944} C_VEL
LIN {X 0,Y 516.886,Z 393.602,A -85,B 0,C 180,E1 -5080.742,E2 -5080.742} C_VEL
LIN {X 0,Y 516.884,Z 393.603,A -85,B 0,C 180,E1 -5082.832,E2 -5082.832} C_VEL
LIN {X 0,Y 516.883,Z 393.602,A -85,B 0,C 180,E1 -5083.904,E2 -5083.904} C_VEL
LIN {X 0,Y 517.014,Z 394.164,A -85,B 0,C 180,E1 -5085.021,E2 -5085.021} C_VEL
LIN {X 0,Y 517.439,Z 397.19,A -85,B 0,C 180,E1 -5087.226,E2 -5087.226} C_VEL
LIN {X 0,Y 517.598,Z 400.317,A -85,B 0,C 180,E1 -5089.327,E2 -5089.327} C_VEL
LIN {X 0,Y 517.41,Z 405.159,A -85,B 0,C 180,E1 -5092.321,E2 -5092.321} C_VEL
LIN {X 0,Y 517.161,Z 410.155,A -85,B 0,C 180,E1 -5095.197,E2 -5095.197} C_VEL
LIN {X 0,Y 517.017,Z 415.329,A -85,B 0,C 180,E1 -5097.985,E2 -5097.985} C_VEL
LIN {X 0,Y 516.912,Z 420.591,A -85,B 0,C 180,E1 -5100.695,E2 -5100.695} C_VEL
LIN {X 0,Y 516.745,Z 426.97,A -85,B 0,C 180,E1 -5103.85,E2 -5103.85} C_VEL
LIN {X 0,Y 516.613,Z 433.088,A -85,B 0,C 180,E1 -5106.764,E2 -5106.764} C_VEL
LIN {X 0,Y 516.572,Z 439.685,A -85,B 0,C 180,E1 -5109.844,E2 -5109.844} C_VEL
LIN {X 0,Y 516.433,Z 445.664,A -85,B 0,C 180,E1 -5112.579,E2 -5112.579} C_VEL
LIN {X 0,Y 516.389,Z 452.85,A -85,B 0,C 180,E1 -5115.82,E2 -5115.82} C_VEL
LIN {X 0,Y 516.394,Z 453.523,A -85,B 0,C 180,E1 -5116.121,E2 -5116.121} C_VEL
LIN {X 0,Y 518.462,Z 465.753,A -85,B 0,C 180,E1 -5116.477,E2 -5116.477} C_VEL
LIN {X 0,Y 518.271,Z 478.161,A -85,B 0,C 180,E1 -5116.921,E2 -5116.921} C_VEL
LIN {X 0,Y 517.976,Z 490.374,A -85,B 0,C 180,E1 -5117.53,E2 -5117.53} C_VEL
LIN {X 0,Y 517.701,Z 500.468,A -85,B 0,C 180,E1 -5118.175,E2 -5118.175} C_VEL
LIN {X 0,Y 517.413,Z 510.186,A -85,B 0,C 180,E1 -5118.939,E2 -5118.939} C_VEL
LIN {X 0,Y 517.174,Z 517.551,A -85,B 0,C 180,E1 -5119.627,E2 -5119.627} C_VEL
LIN {X 0,Y 516.958,Z 524.737,A -85,B 0,C 180,E1 -5120.413,E2 -5120.413} C_VEL
LIN {X 0,Y 516.755,Z 532.283,A -85,B 0,C 180,E1 -5121.396,E2 -5121.396} C_VEL
LIN {X 0,Y 516.563,Z 538.573,A -85,B 0,C 180,E1 -5122.377,E2 -5122.377} C_VEL
LIN {X 0,Y 516.437,Z 544.162,A -85,B 0,C 180,E1 -5123.431,E2 -5123.431} C_VEL
LIN {X 0,Y 516.403,Z 548.903,A -85,B 0,C 180,E1 -5124.533,E2 -5124.533} C_VEL
LIN {X 0,Y 516.343,Z 552.857,A -85,B 0,C 180,E1 -5125.707,E2 -5125.707} C_VEL
LIN {X 0,Y 516.283,Z 555.777,A -85,B 0,C 180,E1 -5126.879,E2 -5126.879} C_VEL
LIN {X 0,Y 516.192,Z 558.194,A -85,B 0,C 180,E1 -5128.439,E2 -5128.439} C_VEL
LIN {X 0,Y 516.16,Z 558.78,A -85,B 0,C 180,E1 -5129.22,E2 -5129.22} C_VEL
LIN {X 0,Y 516.16,Z 558.781,A -85,B 0,C 180,E1 -5130.78,E2 -5130.78} C_VEL
LIN {X 0,Y 516.192,Z 558.195,A -85,B 0,C 180,E1 -5131.56,E2 -5131.56} C_VEL
LIN {X 0,Y 516.282,Z 555.777,A -85,B 0,C 180,E1 -5133.121,E2 -5133.121} C_VEL
LIN {X 0,Y 516.343,Z 552.858,A -85,B 0,C 180,E1 -5134.293,E2 -5134.293} C_VEL
LIN {X 0,Y 516.403,Z 548.904,A -85,B 0,C 180,E1 -5135.466,E2 -5135.466} C_VEL
LIN {X 0,Y 516.443,Z 544.133,A -85,B 0,C 180,E1 -5136.575,E2 -5136.575} C_VEL
LIN {X 0,Y 516.562,Z 538.575,A -85,B 0,C 180,E1 -5137.623,E2 -5137.623} C_VEL
LIN {X 0,Y 516.755,Z 532.285,A -85,B 0,C 180,E1 -5138.604,E2 -5138.604} C_VEL
LIN {X 0,Y 516.957,Z 524.74,A -85,B 0,C 180,E1 -5139.586,E2 -5139.586} C_VEL
LIN {X 0,Y 517.241,Z 515.628,A -85,B 0,C 180,E1 -5140.569,E2 -5140.569} C_VEL
LIN {X 0,Y 517.589,Z 504.191,A -85,B 0,C 180,E1 -5141.553,E2 -5141.553} C_VEL
LIN {X 0,Y 517.821,Z 493.937,A -85,B 0,C 180,E1 -5142.256,E2 -5142.256} C_VEL
LIN {X 0,Y 518.095,Z 483.412,A -85,B 0,C 180,E1 -5142.834,E2 -5142.834} C_VEL
LIN {X 0,Y 518.343,Z 473.069,A -85,B 0,C 180,E1 -5143.276,E2 -5143.276} C_VEL
LIN {X 0,Y 518.301,Z 464.891,A -85,B 0,C 180,E1 -5143.552,E2 -5143.552} C_VEL
LIN {X 0,Y 516.398,Z 453.524,A -85,B 0,C 180,E1 -5143.878,E2 -5143.878} C_VEL
LIN {X 0,Y 516.375,Z 447.461,A -85,B 0,C 180,E1 -5146.607,E2 -5146.607} C_VEL
LIN {X 0,Y 516.484,Z 442.071,A -85,B 0,C 180,E1 -5149.061,E2 -5149.061} C_VEL
LIN {X 0,Y 516.575,Z 436.682,A -85,B 0,C 180,E1 -5151.551,E2 -5151.551} C_VEL
LIN {X 0,Y 516.672,Z 430.826,A -85,B 0,C 180,E1 -5154.305,E2 -5154.305} C_VEL
LIN {X 0,Y 516.806,Z 424.1,A -85,B 0,C 180,E1 -5157.539,E2 -5157.539} C_VEL
LIN {X 0,Y 516.931,Z 418.838,A -85,B 0,C 180,E1 -5160.2,E2 -5160.2} C_VEL
LIN {X 0,Y 517.086,Z 413.575,A -85,B 0,C 180,E1 -5162.933,E2 -5162.933} C_VEL
LIN {X 0,Y 517.214,Z 408.453,A -85,B 0,C 180,E1 -5165.752,E2 -5165.752} C_VEL
LIN {X 0,Y 517.482,Z 403.512,A -85,B 0,C 180,E1 -5168.662,E2 -5168.662} C_VEL
LIN {X 0,Y 517.607,Z 398.758,A -85,B 0,C 180,E1 -5171.687,E2 -5171.687} C_VEL
LIN {X 0,Y 517.199,Z 395.576,A -85,B 0,C 180,E1 -5173.929,E2 -5173.929} C_VEL
LIN {X 0,Y 516.981,Z 394.112,A -85,B 0,C 180,E1 -5175.016,E2 -5175.016} C_VEL
LIN {X 0,Y 516.88,Z 393.6,A -85,B 0,C 180,E1 -5176.106,E2 -5176.106} C_VEL
LIN {X 0,Y 516.915,Z 393.596,A -85,B 0,C 180,E1 -5178.397,E2 -5178.397} C_VEL
LIN {X 0,Y 516.881,Z 393.602,A -85,B 0,C 180,E1 -5181.284,E2 -5181.284} C_VEL
LIN {X 0,Y 516.888,Z 393.598,A -85,B 0,C 180,E1 -5184.221,E2 -5184.221} C_VEL
LIN {X 0,Y 516.894,Z 393.6,A -85,B 0,C 180,E1 -5187.053,E2 -5187.053} C_VEL
LIN {X 0,Y 516.898,Z 393.593,A -85,B 0,C 180,E1 -5189.796,E2 -5189.796} C_VEL
LIN {X 0,Y 516.925,Z 393.593,A -85,B 0,C 180,E1 -5192.467,E2 -5192.467} C_VEL
LIN {X 0,Y 516.906,Z 393.596,A -85,B 0,C 180,E1 -5195.071,E2 -5195.071} C_VEL
LIN {X 0,Y 516.864,Z 393.597,A -85,B 0,C 180,E1 -5197.621,E2 -5197.621} C_VEL
LIN {X 0,Y 516.927,Z 393.591,A -85,B 0,C 180,E1 -5200.129,E2 -5200.129} C_VEL
LIN {X 0,Y 516.926,Z 393.598,A -85,B 0,C 180,E1 -5202.596,E2 -5202.596} C_VEL
LIN {X 0,Y 516.936,Z 393.591,A -85,B 0,C 180,E1 -5205.03,E2 -5205.03} C_VEL
LIN {X 0,Y 516.959,Z 393.589,A -85,B 0,C 180,E1 -5208.233,E2 -5208.233} C_VEL
LIN {X 0,Y 516.964,Z 393.585,A -85,B 0,C 180,E1 -5211.399,E2 -5211.399} C_VEL
LIN {X 0,Y 517.005,Z 393.58,A -85,B 0,C 180,E1 -5213.756,E2 -5213.756} C_VEL
LIN {X 0,Y 517.078,Z 393.571,A -85,B 0,C 180,E1 -5217.663,E2 -5217.663} C_VEL
LIN {X 0,Y 517.088,Z 393.572,A -85,B 0,C 180,E1 -5220.778,E2 -5220.778} C_VEL
LIN {X 0,Y 517.009,Z 393.579,A -85,B 0,C 180,E1 -5223.117,E2 -5223.117} C_VEL
LIN {X 0,Y 517.004,Z 393.588,A -85,B 0,C 180,E1 -5226.243,E2 -5226.243} C_VEL
LIN {X 0,Y 516.948,Z 393.587,A -85,B 0,C 180,E1 -5229.389,E2 -5229.389} C_VEL
LIN {X 0,Y 516.944,Z 393.59,A -85,B 0,C 180,E1 -5231.807,E2 -5231.807} C_VEL
LIN {X 0,Y 516.936,Z 393.588,A -85,B 0,C 180,E1 -5235.146,E2 -5235.146} C_VEL
LIN {X 0,Y 516.918,Z 393.598,A -85,B 0,C 180,E1 -5238.222,E2 -5238.222} C_VEL
LIN {X 0,Y 516.904,Z 393.593,A -85,B 0,C 180,E1 -5240.701,E2 -5240.701} C_VEL
LIN {X 0,Y 516.903,Z 393.601,A -85,B 0,C 180,E1 -5244.072,E2 -5244.072} C_VEL
LIN {X 0,Y 516.922,Z 393.591,A -85,B 0,C 180,E1 -5246.657,E2 -5246.657} C_VEL
LIN {X 0,Y 516.917,Z 393.594,A -85,B 0,C 180,E1 -5249.527,E2 -5249.527} C_VEL
LIN {X 0,Y 516.894,Z 393.594,A -85,B 0,C 180,E1 -5252.545,E2 -5252.545} C_VEL
LIN {X 0,Y 516.876,Z 393.598,A -85,B 0,C 180,E1 -5255.333,E2 -5255.333} C_VEL
LIN {X 0,Y 516.875,Z 393.603,A -85,B 0,C 180,E1 -5257.944,E2 -5257.944} C_VEL
LIN {X 0,Y 516.897,Z 393.593,A -85,B 0,C 180,E1 -5260.74,E2 -5260.74} C_VEL
LIN {X 0,Y 516.875,Z 393.602,A -85,B 0,C 180,E1 -5263.903,E2 -5263.903} C_VEL
LIN {X 0,Y 516.876,Z 393.599,A -85,B 0,C 180,E1 -5266.107,E2 -5266.107} C_VEL
LIN {X 0,Y 516.897,Z 393.597,A -85,B 0,C 180,E1 -5269.261,E2 -5269.261} C_VEL
LIN {X 0,Y 516.895,Z 393.594,A -85,B 0,C 180,E1 -5270.307,E2 -5270.307} C_VEL
LIN {X 0,Y 516.215,Z 393.68,A -85,B 0,C 180,E1 -5270.957,E2 -5270.957} C_VEL
LIN {X 0,Y 513.361,Z 394.042,A -85,B 0,C 180,E1 -5272.012,E2 -5272.012} C_VEL
LIN {X 0,Y 510.954,Z 394.346,A -85,B 0,C 180,E1 -5272.863,E2 -5272.863} C_VEL
LIN {X 0,Y 509.914,Z 394.472,A -85,B 0,C 180,E1 -5273.519,E2 -5273.519} C_VEL
LIN {X 0,Y 509.826,Z 394.48,A -85,B 0,C 180,E1 -5273.741,E2 -5273.741} C_VEL
LIN {X 0,Y 509.858,Z 394.47,A -85,B 0,C 180,E1 -5276.54,E2 -5276.54} C_VEL
LIN {X 0,Y 509.84,Z 394.479,A -85,B 0,C 180,E1 -5279.335,E2 -5279.335} C_VEL
LIN {X 0,Y 509.89,Z 394.467,A -85,B 0,C 180,E1 -5282.055,E2 -5282.055} C_VEL
LIN {X 0,Y 509.873,Z 394.469,A -85,B 0,C 180,E1 -5284.704,E2 -5284.704} C_VEL
LIN {X 0,Y 509.852,Z 394.478,A -85,B 0,C 180,E1 -5287.45,E2 -5287.45} C_VEL
LIN {X 0,Y 509.912,Z 394.465,A -85,B 0,C 180,E1 -5289.845,E2 -5289.845} C_VEL
LIN {X 0,Y 509.88,Z 394.476,A -85,B 0,C 180,E1 -5293.175,E2 -5293.175} C_VEL
LIN {X 0,Y 509.86,Z 394.475,A -85,B 0,C 180,E1 -5295.634,E2 -5295.634} C_VEL
LIN {X 0,Y 509.91,Z 394.469,A -85,B 0,C 180,E1 -5298.875,E2 -5298.875} C_VEL
LIN {X 0,Y 509.948,Z 394.461,A -85,B 0,C 180,E1 -5302.079,E2 -5302.079} C_VEL
LIN {X 0,Y 509.983,Z 394.458,A -85,B 0,C 180,E1 -5304.465,E2 -5304.465} C_VEL
LIN {X 0,Y 510.053,Z 394.449,A -85,B 0,C 180,E1 -5307.631,E2 -5307.631} C_VEL
LIN {X 0,Y 510.061,Z 394.452,A -85,B 0,C 180,E1 -5310.79,E2 -5310.79} C_VEL
LIN {X 0,Y 509.953,Z 394.466,A -85,B 0,C 180,E1 -5313.16,E2 -5313.16} C_VEL
LIN {X 0,Y 509.981,Z 394.459,A -85,B 0,C 180,E1 -5316.33,E2 -5316.33} C_VEL
LIN {X 0,Y 509.914,Z 394.471,A -85,B 0,C 180,E1 -5318.72,E2 -5318.72} C_VEL
LIN {X 0,Y 509.901,Z 394.466,A -85,B 0,C 180,E1 -5321.932,E2 -5321.932} C_VEL
LIN {X 0,Y 509.89,Z 394.47,A -85,B 0,C 180,E1 -5325.242,E2 -5325.242} C_VEL
LIN {X 0,Y 509.885,Z 394.469,A -85,B 0,C 180,E1 -5328.001,E2 -5328.001} C_VEL
LIN {X 0,Y 509.847,Z 394.475,A -85,B 0,C 180,E1 -5331.002,E2 -5331.002} C_VEL
LIN {X 0,Y 509.833,Z 394.473,A -85,B 0,C 180,E1 -5333.563,E2 -5333.563} C_VEL
LIN {X 0,Y 509.91,Z 394.469,A -85,B 0,C 180,E1 -5336.379,E2 -5336.379} C_VEL
LIN {X 0,Y 509.873,Z 394.473,A -85,B 0,C 180,E1 -5338.844,E2 -5338.844} C_VEL
LIN {X 0,Y 509.821,Z 394.474,A -85,B 0,C 180,E1 -5341.59,E2 -5341.59} C_VEL
LIN {X 0,Y 509.849,Z 394.479,A -85,B 0,C 180,E1 -5344.413,E2 -5344.413} C_VEL
LIN {X 0,Y 509.815,Z 394.475,A -85,B 0,C 180,E1 -5347.341,E2 -5347.341} C_VEL
LIN {X 0,Y 509.857,Z 394.479,A -85,B 0,C 180,E1 -5350.38,E2 -5350.38} C_VEL
LIN {X 0,Y 509.835,Z 394.473,A -85,B 0,C 180,E1 -5353.064,E2 -5353.064} C_VEL
LIN {X 0,Y 509.825,Z 394.476,A -85,B 0,C 180,E1 -5355.792,E2 -5355.792} C_VEL
LIN {X 0,Y 509.853,Z 394.475,A -85,B 0,C 180,E1 -5358.575,E2 -5358.575} C_VEL
LIN {X 0,Y 509.847,Z 394.474,A -85,B 0,C 180,E1 -5361.786,E2 -5361.786} C_VEL
LIN {X 0,Y 509.841,Z 394.474,A -85,B 0,C 180,E1 -5364.623,E2 -5364.623} C_VEL
LIN {X 0,Y 509.861,Z 394.471,A -85,B 0,C 180,E1 -5367.481,E2 -5367.481} C_VEL
LIN {X 0,Y 509.877,Z 394.473,A -85,B 0,C 180,E1 -5370.269,E2 -5370.269} C_VEL
LIN {X 0,Y 509.881,Z 394.467,A -85,B 0,C 180,E1 -5372.945,E2 -5372.945} C_VEL
LIN {X 0,Y 509.864,Z 394.472,A -85,B 0,C 180,E1 -5375.574,E2 -5375.574} C_VEL
LIN {X 0,Y 509.817,Z 394.481,A -85,B 0,C 180,E1 -5378.149,E2 -5378.149} C_VEL
LIN {X 0,Y 509.86,Z 394.47,A -85,B 0,C 180,E1 -5380.682,E2 -5380.682} C_VEL
LIN {X 0,Y 509.882,Z 394.468,A -85,B 0,C 180,E1 -5383.175,E2 -5383.175} C_VEL
LIN {X 0,Y 509.86,Z 394.475,A -85,B 0,C 180,E1 -5385.634,E2 -5385.634} C_VEL
LIN {X 0,Y 509.909,Z 394.463,A -85,B 0,C 180,E1 -5388.875,E2 -5388.875} C_VEL
LIN {X 0,Y 509.947,Z 394.463,A -85,B 0,C 180,E1 -5392.079,E2 -5392.079} C_VEL
LIN {X 0,Y 509.979,Z 394.455,A -85,B 0,C 180,E1 -5394.465,E2 -5394.465} C_VEL
LIN {X 0,Y 510.051,Z 394.455,A -85,B 0,C 180,E1 -5397.631,E2 -5397.631} C_VEL
LIN {X 0,Y 510.061,Z 394.445,A -85,B 0,C 180,E1 -5400.79,E2 -5400.79} C_VEL
LIN {X 0,Y 509.954,Z 394.461,A -85,B 0,C 180,E1 -5403.161,E2 -5403.161} C_VEL
LIN {X 0,Y 509.975,Z 394.455,A -85,B 0,C 180,E1 -5406.33,E2 -5406.33} C_VEL
LIN {X 0,Y 509.913,Z 394.463,A -85,B 0,C 180,E1 -5408.721,E2 -5408.721} C_VEL
LIN {X 0,Y 509.901,Z 394.467,A -85,B 0,C 180,E1 -5411.932,E2 -5411.932} C_VEL
LIN {X 0,Y 509.891,Z 394.473,A -85,B 0,C 180,E1 -5415.242,E2 -5415.242} C_VEL
LIN {X 0,Y 509.886,Z 394.467,A -85,B 0,C 180,E1 -5418.002,E2 -5418.002} C_VEL
LIN {X 0,Y 509.848,Z 394.476,A -85,B 0,C 180,E1 -5421.002,E2 -5421.002} C_VEL
LIN {X 0,Y 509.868,Z 394.469,A -85,B 0,C 180,E1 -5424.427,E2 -5424.427} C_VEL
LIN {X 0,Y 509.884,Z 394.474,A -85,B 0,C 180,E1 -5427.056,E2 -5427.056} C_VEL
LIN {X 0,Y 509.856,Z 394.471,A -85,B 0,C 180,E1 -5429.752,E2 -5429.752} C_VEL
LIN {X 0,Y 509.875,Z 394.472,A -85,B 0,C 180,E1 -5432.775,E2 -5432.775} C_VEL
LIN {X 0,Y 509.842,Z 394.476,A -85,B 0,C 180,E1 -5435.582,E2 -5435.582} C_VEL
LIN {X 0,Y 509.85,Z 394.474,A -85,B 0,C 180,E1 -5438.338,E2 -5438.338} C_VEL
LIN {X 0,Y 509.858,Z 394.477,A -85,B 0,C 180,E1 -5441.426,E2 -5441.426} C_VEL
LIN {X 0,Y 509.832,Z 394.481,A -85,B 0,C 180,E1 -5444.208,E2 -5444.208} C_VEL
LIN {X 0,Y 510.358,Z 397.936,A -85,B 0,C 180,E1 -5446.874,E2 -5446.874} C_VEL
LIN {X 0,Y 510.613,Z 401.323,A -85,B 0,C 180,E1 -5449.202,E2 -5449.202} C_VEL
LIN {X 0,Y 510.459,Z 405.275,A -85,B 0,C 180,E1 -5451.716,E2 -5451.716} C_VEL
LIN {X 0,Y 510.182,Z 410.258,A -85,B 0,C 180,E1 -5454.65,E2 -5454.65} C_VEL
LIN {X 0,Y 510.005,Z 415.337,A -85,B 0,C 180,E1 -5457.491,E2 -5457.491} C_VEL
LIN {X 0,Y 509.861,Z 420.635,A -85,B 0,C 180,E1 -5460.274,E2 -5460.274} C_VEL
LIN {X 0,Y 509.706,Z 427.353,A -85,B 0,C 180,E1 -5463.669,E2 -5463.669} C_VEL
LIN {X 0,Y 509.553,Z 433.088,A -85,B 0,C 180,E1 -5466.423,E2 -5466.423} C_VEL
LIN {X 0,Y 509.493,Z 438.478,A -85,B 0,C 180,E1 -5468.983,E2 -5468.983} C_VEL
LIN {X 0,Y 509.376,Z 443.867,A -85,B 0,C 180,E1 -5471.498,E2 -5471.498} C_VEL
LIN {X 0,Y 509.321,Z 451.053,A -85,B 0,C 180,E1 -5474.801,E2 -5474.801} C_VEL
LIN {X 0,Y 509.301,Z 453.523,A -85,B 0,C 180,E1 -5475.924,E2 -5475.924} C_VEL
LIN {X 0,Y 511.408,Z 465.737,A -85,B 0,C 180,E1 -5476.287,E2 -5476.287} C_VEL
LIN {X 0,Y 511.349,Z 478.161,A -85,B 0,C 180,E1 -5476.741,E2 -5476.741} C_VEL
LIN {X 0,Y 511.039,Z 490.384,A -85,B 0,C 180,E1 -5477.359,E2 -5477.359} C_VEL
LIN {X 0,Y 510.754,Z 499.833,A -85,B 0,C 180,E1 -5477.965,E2 -5477.965} C_VEL
LIN {X 0,Y 510.435,Z 510.179,A -85,B 0,C 180,E1 -5478.786,E2 -5478.786} C_VEL
LIN {X 0,Y 510.182,Z 517.545,A -85,B 0,C 180,E1 -5479.483,E2 -5479.483} C_VEL
LIN {X 0,Y 509.953,Z 524.733,A -85,B 0,C 180,E1 -5480.28,E2 -5480.28} C_VEL
LIN {X 0,Y 509.72,Z 532.278,A -85,B 0,C 180,E1 -5481.276,E2 -5481.276} C_VEL
LIN {X 0,Y 509.522,Z 538.568,A -85,B 0,C 180,E1 -5482.271,E2 -5482.271} C_VEL
LIN {X 0,Y 509.35,Z 544.656,A -85,B 0,C 180,E1 -5483.443,E2 -5483.443} C_VEL
LIN {X 0,Y 509.247,Z 550.385,A -85,B 0,C 180,E1 -5484.853,E2 -5484.853} C_VEL
LIN {X 0,Y 509.253,Z 553.974,A -85,B 0,C 180,E1 -5486.043,E2 -5486.043} C_VEL
LIN {X 0,Y 509.201,Z 555.774,A -85,B 0,C 180,E1 -5486.835,E2 -5486.835} C_VEL
LIN {X 0,Y 509.113,Z 558.195,A -85,B 0,C 180,E1 -5488.418,E2 -5488.418} C_VEL
LIN {X 0,Y 509.074,Z 558.78,A -85,B 0,C 180,E1 -5489.209,E2 -5489.209} C_VEL
LIN {X 0,Y 509.074,Z 558.78,A -85,B 0,C 180,E1 -5490.791,E2 -5490.791} C_VEL
LIN {X 0,Y 509.113,Z 558.196,A -85,B 0,C 180,E1 -5491.582,E2 -5491.582} C_VEL
LIN {X 0,Y 509.201,Z 555.775,A -85,B 0,C 180,E1 -5493.165,E2 -5493.165} C_VEL
LIN {X 0,Y 509.233,Z 552.855,A -85,B 0,C 180,E1 -5494.353,E2 -5494.353} C_VEL
LIN {X 0,Y 509.342,Z 548.9,A -85,B 0,C 180,E1 -5495.542,E2 -5495.542} C_VEL
LIN {X 0,Y 509.404,Z 543.278,A -85,B 0,C 180,E1 -5496.844,E2 -5496.844} C_VEL
LIN {X 0,Y 509.585,Z 536.256,A -85,B 0,C 180,E1 -5498.126,E2 -5498.126} C_VEL
LIN {X 0,Y 509.85,Z 527.977,A -85,B 0,C 180,E1 -5499.321,E2 -5499.321} C_VEL
LIN {X 0,Y 510.068,Z 519.461,A -85,B 0,C 180,E1 -5500.318,E2 -5500.318} C_VEL
LIN {X 0,Y 510.408,Z 511.315,A -85,B 0,C 180,E1 -5501.114,E2 -5501.114} C_VEL
LIN {X 0,Y 510.674,Z 502.835,A -85,B 0,C 180,E1 -5501.812,E2 -5501.812} C_VEL
LIN {X 0,Y 510.884,Z 493.945,A -85,B 0,C 180,E1 -5502.424,E2 -5502.424} C_VEL
LIN {X 0,Y 511.153,Z 483.402,A -85,B 0,C 180,E1 -5503.011,E2 -5503.011} C_VEL
LIN {X 0,Y 511.422,Z 473.059,A -85,B 0,C 180,E1 -5503.459,E2 -5503.459} C_VEL
LIN {X 0,Y 511.409,Z 465.749,A -85,B 0,C 180,E1 -5503.712,E2 -5503.712} C_VEL
LIN {X 0,Y 509.444,Z 454.619,A -85,B 0,C 180,E1 -5504.046,E2 -5504.046} C_VEL
LIN {X 0,Y 509.304,Z 453.524,A -85,B 0,C 180,E1 -5504.076,E2 -5504.076} C_VEL
LIN {X 0,Y 509.312,Z 447.461,A -85,B 0,C 180,E1 -5506.844,E2 -5506.844} C_VEL
LIN {X 0,Y 509.51,Z 440.275,A -85,B 0,C 180,E1 -5510.172,E2 -5510.172} C_VEL
LIN {X 0,Y 509.543,Z 434.885,A -85,B 0,C 180,E1 -5512.718,E2 -5512.718} C_VEL
LIN {X 0,Y 509.63,Z 429.496,A -85,B 0,C 180,E1 -5515.309,E2 -5515.309} C_VEL
LIN {X 0,Y 509.742,Z 423.875,A -85,B 0,C 180,E1 -5518.067,E2 -5518.067} C_VEL
LIN {X 0,Y 509.901,Z 418.835,A -85,B 0,C 180,E1 -5520.661,E2 -5520.661} C_VEL
LIN {X 0,Y 510.087,Z 413.603,A -85,B 0,C 180,E1 -5523.443,E2 -5523.443} C_VEL
LIN {X 0,Y 510.226,Z 408.559,A -85,B 0,C 180,E1 -5526.319,E2 -5526.319} C_VEL
LIN {X 0,Y 510.523,Z 403.647,A -85,B 0,C 180,E1 -5529.289,E2 -5529.289} C_VEL
LIN {X 0,Y 510.604,Z 400.459,A -85,B 0,C 180,E1 -5531.35,E2 -5531.35} C_VEL
LIN {X 0,Y 510.276,Z 397.394,A -85,B 0,C 180,E1 -5533.522,E2 -5533.522} C_VEL
LIN {X 0,Y 509.829,Z 394.48,A -85,B 0,C 180,E1 -5535.791,E2 -5535.791} C_VEL
LIN {X 0,Y 509.856,Z 394.477,A -85,B 0,C 180,E1 -5538.574,E2 -5538.574} C_VEL
LIN {X 0,Y 509.849,Z 394.474,A -85,B 0,C 180,E1 -5541.785,E2 -5541.785} C_VEL
LIN {X 0,Y 509.843,Z 394.479,A -85,B 0,C 180,E1 -5544.623,E2 -5544.623} C_VEL
LIN {X 0,Y 509.862,Z 394.471,A -85,B 0,C 180,E1 -5547.48,E2 -5547.48} C_VEL
LIN {X 0,Y 509.878,Z 394.469,A -85,B 0,C 180,E1 -5550.268,E2 -5550.268} C_VEL
LIN {X 0,Y 509.882,Z 394.474,A -85,B 0,C 180,E1 -5552.944,E2 -5552.944} C_VEL
LIN {X 0,Y 509.865,Z 394.469,A -85,B 0,C 180,E1 -5555.573,E2 -5555.573} C_VEL
LIN {X 0,Y 509.845,Z 394.476,A -85,B 0,C 180,E1 -5558.998,E2 -5558.998} C_VEL
LIN {X 0,Y 509.883,Z 394.468,A -85,B 0,C 180,E1 -5561.998,E2 -5561.998} C_VEL
LIN {X 0,Y 509.904,Z 394.47,A -85,B 0,C 180,E1 -5564.818,E2 -5564.818} C_VEL
LIN {X 0,Y 509.895,Z 394.468,A -85,B 0,C 180,E1 -5568.123,E2 -5568.123} C_VEL
LIN {X 0,Y 509.911,Z 394.464,A -85,B 0,C 180,E1 -5571.279,E2 -5571.279} C_VEL
LIN {X 0,Y 509.973,Z 394.456,A -85,B 0,C 180,E1 -5573.67,E2 -5573.67} C_VEL
LIN {X 0,Y 510.049,Z 394.446,A -85,B 0,C 180,E1 -5577.63,E2 -5577.63} C_VEL
LIN {X 0,Y 510.058,Z 394.448,A -85,B 0,C 180,E1 -5580.789,E2 -5580.789} C_VEL
LIN {X 0,Y 509.951,Z 394.458,A -85,B 0,C 180,E1 -5583.16,E2 -5583.16} C_VEL
LIN {X 0,Y 509.972,Z 394.464,A -85,B 0,C 180,E1 -5586.329,E2 -5586.329} C_VEL
LIN {X 0,Y 509.91,Z 394.466,A -85,B 0,C 180,E1 -5588.72,E2 -5588.72} C_VEL
LIN {X 0,Y 509.896,Z 394.47,A -85,B 0,C 180,E1 -5591.931,E2 -5591.931} C_VEL
LIN {X 0,Y 509.886,Z 394.466,A -85,B 0,C 180,E1 -5595.242,E2 -5595.242} C_VEL
LIN {X 0,Y 509.881,Z 394.474,A -85,B 0,C 180,E1 -5598.001,E2 -5598.001} C_VEL
LIN {X 0,Y 509.842,Z 394.472,A -85,B 0,C 180,E1 -5601.002,E2 -5601.002} C_VEL
LIN {X 0,Y 509.829,Z 394.476,A -85,B 0,C 180,E1 -5603.563,E2 -5603.563} C_VEL
LIN {X 0,Y 509.906,Z 394.467,A -85,B 0,C 180,E1 -5606.379,E2 -5606.379} C_VEL
LIN {X 0,Y 509.878,Z 394.467,A -85,B 0,C 180,E1 -5608.844,E2 -5608.844} C_VEL
LIN {X 0,Y 509.819,Z 394.479,A -85,B 0,C 180,E1 -5611.59,E2 -5611.59} C_VEL
LIN {X 0,Y 509.847,Z 394.473,A -85,B 0,C 180,E1 -5614.413,E2 -5614.413} C_VEL
LIN {X 0,Y 509.812,Z 394.478,A -85,B 0,C 180,E1 -5617.341,E2 -5617.341} C_VEL
LIN {X 0,Y 509.854,Z 394.472,A -85,B 0,C 180,E1 -5620.38,E2 -5620.38} C_VEL
LIN {X 0,Y 509.832,Z 394.474,A -85,B 0,C 180,E1 -5623.064,E2 -5623.064} C_VEL
LIN {X 0,Y 509.824,Z 394.481,A -85,B 0,C 180,E1 -5625.792,E2 -5625.792} C_VEL
LIN {X 0,Y 509.859,Z 394.47,A -85,B 0,C 180,E1 -5628.576,E2 -5628.576} C_VEL
LIN {X 0,Y 509.846,Z 394.477,A -85,B 0,C 180,E1 -5631.786,E2 -5631.786} C_VEL
